C01810=1224.930,186.137,-55.083,-177.570,5.975,148.343
C01811=1224.935,185.867,-55.058,-177.573,5.973,148.343
C01812=1224.941,185.598,-55.033,-177.576,5.971,148.344
C01813=1224.945,185.328,-55.009,-177.578,5.969,148.344
C01814=1224.951,185.058,-54.984,-177.580,5.968,148.345
C01815=1224.955,184.810,-54.961,-177.584,5.967,148.345
C01816=1224.959,184.561,-54.938,-177.586,5.965,148.345
C01817=1224.964,184.311,-54.915,-177.589,5.963,148.346
C01818=1224.969,184.063,-54.893,-177.591,5.962,148.346
C01819=1224.974,183.814,-54.869,-177.594,5.960,148.347
C01820=1224.978,183.565,-54.846,-177.597,5.959,148.347
C01821=1224.982,183.316,-54.823,-177.599,5.958,148.348
C01822=1224.987,183.067,-54.800,-177.602,5.956,148.348
C01823=1224.992,182.819,-54.778,-177.604,5.954,148.348
C01824=1224.997,182.569,-54.755,-177.606,5.953,148.349
C01825=1225.002,182.320,-54.732,-177.609,5.952,148.349
C01826=1225.005,182.071,-54.709,-177.612,5.950,148.350
C01827=1225.011,181.823,-54.686,-177.614,5.949,148.350
C01828=1225.015,181.574,-54.664,-177.617,5.947,148.350
C01829=1225.020,181.324,-54.641,-177.620,5.945,148.351
C01830=1225.024,181.076,-54.618,-177.622,5.944,148.351
C01831=1225.029,180.827,-54.595,-177.625,5.943,148.352
C01832=1225.034,180.578,-54.572,-177.627,5.941,148.352
C01833=1225.038,180.329,-54.550,-177.629,5.940,148.352
C01834=1225.043,180.079,-54.527,-177.633,5.938,148.353
C01835=1225.048,179.831,-54.505,-177.635,5.936,148.353
C01836=1225.052,179.582,-54.481,-177.637,5.935,148.354
C01837=1225.057,179.333,-54.459,-177.640,5.934,148.354
C01838=1225.062,179.085,-54.436,-177.643,5.932,148.355
C01839=1225.066,178.835,-54.414,-177.645,5.931,148.355
C01840=1225.071,178.586,-54.391,-177.648,5.929,148.355
C01841=1225.075,178.338,-54.368,-177.650,5.928,148.356
C01842=1225.080,178.089,-54.346,-177.653,5.926,148.356
C01843=1225.084,177.840,-54.323,-177.656,5.925,148.357
C01844=1225.089,177.590,-54.300,-177.658,5.924,148.357
C01845=1225.094,177.342,-54.278,-177.660,5.922,148.357
C01846=1225.098,177.093,-54.256,-177.663,5.920,148.358
C01847=1225.103,176.844,-54.233,-177.666,5.920,148.358
C01848=1225.108,176.595,-54.211,-177.668,5.918,148.359
C01849=1225.112,176.346,-54.188,-177.671,5.916,148.359
C01850=1225.117,176.097,-54.166,-177.673,5.915,148.359
C01851=1225.122,175.848,-54.143,-177.676,5.913,148.360
C01852=1225.126,175.599,-54.120,-177.678,5.912,148.360
C01853=1225.131,175.350,-54.099,-177.681,5.911,148.361
C01854=1225.136,175.101,-54.075,-177.684,5.909,148.361
C01855=1225.140,174.852,-54.053,-177.686,5.908,148.362
C01856=1225.145,174.604,-54.030,-177.689,5.906,148.362
C01857=1225.150,174.354,-54.008,-177.691,5.904,148.362
C01858=1225.154,174.105,-53.986,-177.694,5.903,148.363
C01859=1225.159,173.857,-53.963,-177.697,5.902,148.363
C01860=1225.164,173.607,-53.941,-177.699,5.901,148.364
C01861=1225.168,173.359,-53.919,-177.701,5.899,148.364
C01862=1225.173,173.110,-53.896,-177.704,5.897,148.365
C01863=1225.177,172.860,-53.874,-177.707,5.897,148.365
C01864=1225.182,172.612,-53.852,-177.709,5.895,148.365
C01865=1225.187,172.363,-53.829,-177.712,5.893,148.366
C01866=1225.192,172.114,-53.807,-177.715,5.892,148.366
C01867=1225.196,171.865,-53.785,-177.717,5.890,148.367
C01868=1225.201,171.616,-53.762,-177.719,5.889,148.367
C01869=1225.206,171.367,-53.740,-177.722,5.888,148.368
C01870=1225.210,171.118,-53.718,-177.725,5.886,148.368
C01871=1225.214,170.870,-53.696,-177.727,5.885,148.369
C01872=1225.219,170.620,-53.673,-177.730,5.883,148.369
C01873=1225.224,170.371,-53.652,-177.732,5.882,148.369
C01874=1225.229,170.122,-53.630,-177.735,5.881,148.370
C01875=1225.233,169.873,-53.607,-177.737,5.880,148.370
C01876=1225.238,169.624,-53.584,-177.740,5.878,148.371
C01877=1225.242,169.375,-53.562,-177.743,5.876,148.371
C01878=1225.247,169.126,-53.541,-177.745,5.875,148.372
C01879=1225.252,168.877,-53.519,-177.748,5.874,148.372
C01880=1225.257,168.628,-53.496,-177.750,5.873,148.372
C01881=1225.261,168.379,-53.474,-177.753,5.871,148.373
C01882=1225.266,168.131,-53.452,-177.756,5.869,148.373
C01883=1225.270,167.881,-53.430,-177.758,5.868,148.374
C01884=1225.275,167.633,-53.408,-177.761,5.867,148.374
C01885=1225.280,167.383,-53.386,-177.763,5.866,148.375
C01886=1225.285,167.134,-53.364,-177.766,5.864,148.375
C01887=1225.289,166.885,-53.342,-177.768,5.863,148.376
C01888=1225.294,166.637,-53.320,-177.771,5.862,148.376
C01889=1225.298,166.387,-53.298,-177.774,5.860,148.376
C01890=1225.303,166.139,-53.276,-177.776,5.859,148.377
C01891=1225.308,165.889,-53.254,-177.779,5.857,148.377
C01892=1225.313,165.640,-53.232,-177.781,5.856,148.378
C01893=1225.317,165.392,-53.209,-177.784,5.854,148.378
C01894=1225.322,165.143,-53.188,-177.786,5.854,148.379
C01895=1225.326,164.894,-53.166,-177.789,5.852,148.379
C01896=1225.331,164.645,-53.144,-177.791,5.850,148.379
C01897=1225.335,164.396,-53.122,-177.794,5.849,148.380
C01898=1225.340,164.147,-53.100,-177.797,5.848,148.380
C01899=1225.345,163.898,-53.079,-177.799,5.847,148.381
C01900=1225.350,163.648,-53.057,-177.802,5.845,148.381
C01901=1225.355,163.399,-53.035,-177.804,5.844,148.382
C01902=1225.360,163.150,-53.013,-177.807,5.842,148.382
C01903=1225.364,162.901,-52.991,-177.809,5.842,148.383
C01904=1225.369,162.652,-52.969,-177.812,5.840,148.383
C01905=1225.374,162.403,-52.947,-177.815,5.838,148.384
C01906=1225.378,162.155,-52.926,-177.817,5.837,148.384
C01907=1225.383,161.905,-52.904,-177.820,5.836,148.384
C01908=1225.388,161.657,-52.882,-177.822,5.835,148.385
C01909=1225.392,161.407,-52.860,-177.825,5.833,148.385
C01910=1225.397,161.159,-52.838,-177.827,5.832,148.386
C01911=1225.402,160.910,-52.817,-177.830,5.830,148.386
C01912=1225.406,160.660,-52.795,-177.832,5.830,148.387
C01913=1225.411,160.412,-52.774,-177.835,5.828,148.387
C01914=1225.415,160.162,-52.752,-177.837,5.827,148.388
C01915=1225.421,159.893,-52.728,-177.840,5.825,148.388
C01916=1225.425,159.624,-52.705,-177.843,5.823,148.389
C01917=1225.431,159.355,-52.681,-177.846,5.822,148.389
C01918=1225.435,159.086,-52.659,-177.848,5.821,148.390
C01919=1225.440,158.837,-52.637,-177.851,5.819,148.390
C01920=1225.445,158.588,-52.615,-177.854,5.818,148.391
C01921=1225.449,158.339,-52.593,-177.856,5.817,148.391
C01922=1225.455,158.090,-52.572,-177.859,5.816,148.392
C01923=1225.459,157.841,-52.550,-177.861,5.814,148.392
C01924=1225.464,157.592,-52.529,-177.864,5.814,148.393
C01925=1225.469,157.343,-52.508,-177.867,5.812,148.393
C01926=1225.473,157.094,-52.486,-177.869,5.811,148.393
C01927=1225.478,156.845,-52.464,-177.872,5.809,148.394
C01928=1225.483,156.596,-52.442,-177.874,5.808,148.394
C01929=1225.487,156.347,-52.421,-177.877,5.806,148.395
C01930=1225.492,156.098,-52.400,-177.879,5.806,148.395
C01931=1225.497,155.849,-52.378,-177.882,5.804,148.396
C01932=1225.502,155.600,-52.357,-177.884,5.803,148.396
C01933=1225.506,155.351,-52.335,-177.887,5.801,148.397
C01934=1225.511,155.101,-52.314,-177.889,5.800,148.397
C01935=1225.516,154.853,-52.292,-177.893,5.799,148.398
C01936=1225.520,154.604,-52.271,-177.895,5.798,148.398
C01937=1225.525,154.355,-52.250,-177.897,5.796,148.398
C01938=1225.530,154.106,-52.228,-177.900,5.796,148.399
C01939=1225.534,153.856,-52.207,-177.903,5.794,148.399
C01940=1225.539,153.607,-52.185,-177.905,5.793,148.400
C01941=1225.544,153.359,-52.164,-177.908,5.791,148.400
C01942=1225.548,153.110,-52.143,-177.910,5.790,148.401
C01943=1225.553,152.860,-52.121,-177.913,5.789,148.401
C01944=1225.558,152.611,-52.100,-177.915,5.788,148.402
C01945=1225.563,152.362,-52.079,-177.918,5.786,148.402
C01946=1225.568,152.113,-52.058,-177.920,5.785,148.403
C01947=1225.571,151.864,-52.036,-177.923,5.783,148.403
C01948=1225.577,151.615,-52.015,-177.926,5.783,148.404
C01949=1225.581,151.366,-51.993,-177.928,5.781,148.404
C01950=1225.587,151.117,-51.972,-177.930,5.780,148.405
C01951=1225.591,150.869,-51.951,-177.934,5.779,148.405
C01952=1225.595,150.619,-51.930,-177.936,5.778,148.406
C01953=1225.600,150.369,-51.909,-177.939,5.776,148.406
C01954=1225.605,150.121,-51.888,-177.941,5.775,148.407
C01955=1225.610,149.872,-51.867,-177.944,5.773,148.407
C01956=1225.614,149.623,-51.845,-177.946,5.773,148.408
C01957=1225.619,149.373,-51.824,-177.949,5.771,148.408
C01958=1225.624,149.124,-51.804,-177.951,5.770,148.409
C01959=1225.629,148.876,-51.782,-177.954,5.769,148.409
C01960=1225.634,148.626,-51.761,-177.956,5.767,148.409
C01961=1225.637,148.377,-51.740,-177.959,5.767,148.410
C01962=1225.642,148.128,-51.719,-177.962,5.765,148.410
C01963=1225.648,147.879,-51.698,-177.964,5.764,148.411
C01964=1225.652,147.631,-51.677,-177.967,5.762,148.411
C01965=1225.657,147.381,-51.656,-177.969,5.761,148.412
C01966=1225.662,147.132,-51.635,-177.972,5.760,148.412
C01967=1225.666,146.883,-51.613,-177.974,5.759,148.413
C01968=1225.671,146.634,-51.592,-177.977,5.758,148.413
C01969=1225.675,146.385,-51.572,-177.979,5.757,148.414
C01970=1225.680,146.136,-51.551,-177.982,5.756,148.414
C01971=1225.685,145.887,-51.529,-177.985,5.754,148.415
C01972=1225.690,145.638,-51.509,-177.987,5.753,148.415
C01973=1225.695,145.389,-51.488,-177.990,5.752,148.416
C01974=1225.699,145.139,-51.467,-177.992,5.751,148.416
C01975=1225.704,144.890,-51.445,-177.995,5.749,148.417
C01976=1225.709,144.641,-51.424,-177.997,5.748,148.417
C01977=1225.713,144.392,-51.404,-178.000,5.748,148.418
C01978=1225.718,144.143,-51.383,-178.003,5.746,148.418
C01979=1225.723,143.894,-51.363,-178.005,5.745,148.418
C01980=1225.728,143.645,-51.341,-178.008,5.743,148.419
C01981=1225.732,143.396,-51.321,-178.010,5.742,148.419
C01982=1225.737,143.147,-51.300,-178.013,5.741,148.420
C01983=1225.741,142.897,-51.279,-178.015,5.740,148.420
C01984=1225.746,142.648,-51.258,-178.018,5.739,148.421
C01985=1225.751,142.399,-51.238,-178.020,5.737,148.421
C01986=1225.756,142.151,-51.216,-178.023,5.737,148.422
C01987=1225.760,141.902,-51.196,-178.026,5.735,148.422
C01988=1225.765,141.652,-51.175,-178.028,5.734,148.423
C01989=1225.770,141.403,-51.154,-178.031,5.732,148.424
C01990=1225.775,141.154,-51.133,-178.033,5.732,148.424
C01991=1225.779,140.905,-51.113,-178.036,5.731,148.425
C01992=1225.784,140.656,-51.092,-178.038,5.729,148.425
C01993=1225.789,140.407,-51.072,-178.041,5.728,148.426
C01994=1225.794,140.158,-51.051,-178.044,5.727,148.426
C01995=1225.798,139.909,-51.030,-178.046,5.726,148.427
C01996=1225.804,139.660,-51.009,-178.048,5.725,148.427
C01997=1225.808,139.411,-50.989,-178.052,5.724,148.428
C01998=1225.812,139.161,-50.968,-178.054,5.723,148.428
C01999=1225.817,138.912,-50.947,-178.056,5.721,148.428
C02000=1225.822,138.663,-50.927,-178.059,5.720,148.429
C02001=1225.827,138.414,-50.906,-178.061,5.719,148.429
C02002=1225.831,138.165,-50.885,-178.064,5.718,148.430
C02003=1225.836,137.915,-50.864,-178.066,5.717,148.430
C02004=1225.841,137.666,-50.844,-178.069,5.715,148.431
C02005=1225.845,137.417,-50.824,-178.072,5.714,148.431
C02006=1225.850,137.168,-50.803,-178.074,5.714,148.432
C02007=1225.855,136.919,-50.782,-178.077,5.712,148.432
C02008=1225.859,136.670,-50.762,-178.079,5.711,148.433
C02009=1225.864,136.421,-50.741,-178.082,5.709,148.433
C02010=1225.869,136.172,-50.721,-178.085,5.709,148.434
C02011=1225.874,135.922,-50.701,-178.087,5.708,148.434
C02012=1225.879,135.673,-50.680,-178.090,5.706,148.435
C02013=1225.883,135.424,-50.660,-178.092,5.705,148.435
C02014=1225.888,135.176,-50.640,-178.095,5.705,148.436
C02015=1225.893,134.927,-50.619,-178.097,5.703,148.436
C02016=1225.898,134.678,-50.598,-178.100,5.702,148.437
C02017=1225.903,134.428,-50.579,-178.103,5.700,148.437
C02018=1225.908,134.179,-50.558,-178.105,5.700,148.438
C02019=1225.912,133.910,-50.536,-178.108,5.698,148.439
C02020=1225.917,133.641,-50.514,-178.111,5.697,148.439
C02021=1225.923,133.373,-50.491,-178.114,5.696,148.440
C02022=1225.928,133.104,-50.470,-178.116,5.695,148.440
C02023=1225.933,132.855,-50.449,-178.119,5.693,148.441
C02024=1225.937,132.606,-50.429,-178.121,5.692,148.441
C02025=1225.942,132.357,-50.409,-178.124,5.692,148.442
C02026=1225.946,132.108,-50.389,-178.126,5.690,148.442
C02027=1225.952,131.858,-50.368,-178.129,5.689,148.443
C02028=1225.956,131.609,-50.348,-178.131,5.688,148.443
C02029=1225.961,131.360,-50.327,-178.134,5.687,148.444
C02030=1225.966,131.112,-50.308,-178.136,5.686,148.444
C02031=1225.971,130.862,-50.287,-178.139,5.685,148.445
C02032=1225.975,130.613,-50.267,-178.142,5.683,148.445
C02033=1225.980,130.364,-50.247,-178.144,5.683,148.446
C02034=1225.985,130.115,-50.227,-178.146,5.682,148.446
C02035=1225.989,129.866,-50.206,-178.150,5.680,148.447
C02036=1225.995,129.616,-50.186,-178.152,5.679,148.447
C02037=1225.999,129.367,-50.166,-178.155,5.678,148.448
C02038=1226.004,129.119,-50.146,-178.157,5.677,148.448
C02039=1226.009,128.869,-50.126,-178.160,5.676,148.449
C02040=1226.013,128.620,-50.106,-178.163,5.675,148.450
C02041=1226.018,128.371,-50.086,-178.165,5.674,148.450
C02042=1226.023,128.121,-50.065,-178.167,5.673,148.451
C02043=1226.028,127.873,-50.045,-178.170,5.672,148.451
C02044=1226.032,127.623,-50.025,-178.173,5.671,148.452
C02045=1226.037,127.375,-50.005,-178.175,5.670,148.452
C02046=1226.042,127.125,-49.985,-178.178,5.668,148.453
C02047=1226.047,126.876,-49.965,-178.180,5.667,148.453
C02048=1226.051,126.627,-49.945,-178.183,5.667,148.454
C02049=1226.056,126.378,-49.925,-178.185,5.665,148.454
C02050=1226.060,126.128,-49.905,-178.188,5.664,148.455
C02051=1226.066,125.880,-49.885,-178.190,5.663,148.455
C02052=1226.071,125.630,-49.865,-178.193,5.662,148.456
C02053=1226.075,125.381,-49.845,-178.195,5.661,148.456
C02054=1226.080,125.131,-49.825,-178.198,5.660,148.457
C02055=1226.085,124.883,-49.805,-178.201,5.660,148.457
C02056=1226.090,124.634,-49.785,-178.203,5.658,148.458
C02057=1226.094,124.385,-49.765,-178.206,5.657,148.458
C02058=1226.099,124.135,-49.745,-178.208,5.656,148.459
C02059=1226.104,123.886,-49.725,-178.211,5.655,148.459
C02060=1226.108,123.637,-49.705,-178.213,5.654,148.460
C02061=1226.114,123.388,-49.686,-178.216,5.653,148.461
C02062=1226.118,123.139,-49.666,-178.219,5.651,148.461
C02063=1226.123,122.889,-49.646,-178.221,5.651,148.462
C02064=1226.127,122.640,-49.626,-178.223,5.650,148.462
C02065=1226.133,122.391,-49.606,-178.226,5.648,148.463
C02066=1226.137,122.142,-49.587,-178.229,5.648,148.463
C02067=1226.142,121.893,-49.566,-178.231,5.647,148.464
C02068=1226.147,121.643,-49.547,-178.234,5.646,148.464
C02069=1226.152,121.394,-49.527,-178.236,5.644,148.465
C02070=1226.156,121.146,-49.507,-178.239,5.644,148.465
C02071=1226.161,120.896,-49.487,-178.241,5.643,148.466
C02072=1226.166,120.646,-49.468,-178.244,5.641,148.466
C02073=1226.171,120.398,-49.448,-178.247,5.641,148.467
C02074=1226.176,120.149,-49.428,-178.249,5.640,148.467
C02075=1226.180,119.899,-49.408,-178.252,5.638,148.468
C02076=1226.186,119.650,-49.389,-178.254,5.637,148.468
C02077=1226.189,119.401,-49.369,-178.257,5.637,148.469
C02078=1226.194,119.152,-49.350,-178.259,5.636,148.469
C02079=1226.199,118.902,-49.330,-178.262,5.634,148.470
C02080=1226.204,118.653,-49.311,-178.265,5.634,148.471
C02081=1226.209,118.405,-49.290,-178.267,5.633,148.471
C02082=1226.213,118.155,-49.271,-178.270,5.631,148.472
C02083=1226.219,117.906,-49.251,-178.272,5.630,148.472
C02084=1226.223,117.657,-49.232,-178.275,5.630,148.473
C02085=1226.228,117.407,-49.212,-178.277,5.629,148.473
C02086=1226.233,117.159,-49.193,-178.280,5.627,148.474
C02087=1226.237,116.909,-49.173,-178.283,5.627,148.474
C02088=1226.242,116.660,-49.153,-178.285,5.626,148.475
C02089=1226.247,116.411,-49.134,-178.288,5.625,148.476
C02090=1226.252,116.161,-49.114,-178.290,5.623,148.476
C02091=1226.257,115.912,-49.095,-178.293,5.623,148.477
C02092=1226.262,115.663,-49.075,-178.295,5.622,148.477
C02093=1226.266,115.414,-49.056,-178.298,5.620,148.478
C02094=1226.271,115.165,-49.036,-178.301,5.620,148.478
C02095=1226.276,114.916,-49.017,-178.303,5.619,148.479
C02096=1226.281,114.666,-48.997,-178.305,5.618,148.479
C02097=1226.286,114.418,-48.978,-178.309,5.617,148.480
C02098=1226.290,114.168,-48.959,-178.311,5.616,148.480
C02099=1226.295,113.919,-48.939,-178.313,5.615,148.481
C02100=1226.300,113.670,-48.920,-178.315,5.614,148.481
C02101=1226.305,113.420,-48.900,-178.319,5.613,148.482
C02102=1226.309,113.171,-48.881,-178.321,5.612,148.483
C02103=1226.314,112.922,-48.862,-178.323,5.611,148.483
C02104=1226.319,112.673,-48.842,-178.326,5.610,148.484
C02105=1226.324,112.424,-48.823,-178.329,5.609,148.484
C02106=1226.328,112.174,-48.804,-178.331,5.608,148.485
C02107=1226.333,111.925,-48.784,-178.334,5.607,148.485
C02108=1226.338,111.676,-48.765,-178.336,5.606,148.486
C02109=1226.343,111.426,-48.745,-178.339,5.605,148.486
C02110=1226.348,111.178,-48.726,-178.341,5.604,148.487
C02111=1226.353,110.928,-48.707,-178.344,5.603,148.487
C02112=1226.358,110.679,-48.687,-178.347,5.603,148.488
C02113=1226.362,110.430,-48.668,-178.349,5.601,148.489
C02114=1226.367,110.181,-48.649,-178.352,5.600,148.489
C02115=1226.372,109.932,-48.629,-178.354,5.600,148.490
C02116=1226.376,109.682,-48.610,-178.357,5.599,148.490
C02117=1226.382,109.433,-48.592,-178.359,5.598,148.491
C02118=1226.386,109.183,-48.572,-178.362,5.596,148.491
C02119=1226.391,108.935,-48.553,-178.364,5.596,148.492
C02120=1226.396,108.685,-48.534,-178.367,5.595,148.493
C02121=1226.401,108.436,-48.514,-178.369,5.594,148.493
C02122=1226.405,108.187,-48.495,-178.372,5.593,148.494
C02123=1226.411,107.919,-48.475,-178.375,5.592,148.494
C02124=1226.416,107.650,-48.454,-178.378,5.591,148.495
C02125=1226.421,107.382,-48.434,-178.380,5.590,148.495
C02126=1226.426,107.113,-48.413,-178.383,5.589,148.496
C02127=1226.431,106.864,-48.395,-178.386,5.588,148.497
C02128=1226.436,106.615,-48.375,-178.389,5.587,148.497
C02129=1226.440,106.366,-48.356,-178.391,5.586,148.498
C02130=1226.445,106.116,-48.337,-178.393,5.585,148.498
C02131=1226.451,105.867,-48.318,-178.396,5.584,148.499
C02132=1226.455,105.618,-48.299,-178.398,5.584,148.499
C02133=1226.460,105.369,-48.280,-178.401,5.582,148.500
C02134=1226.464,105.120,-48.261,-178.404,5.581,148.500
C02135=1226.470,104.870,-48.242,-178.406,5.581,148.501
C02136=1226.474,104.621,-48.223,-178.409,5.580,148.502
C02137=1226.479,104.372,-48.204,-178.411,5.579,148.502
C02138=1226.484,104.122,-48.184,-178.414,5.578,148.503
C02139=1226.489,103.873,-48.166,-178.417,5.577,148.503
C02140=1226.494,103.624,-48.146,-178.419,5.576,148.504
C02141=1226.498,103.375,-48.128,-178.421,5.576,148.504
C02142=1226.503,103.125,-48.109,-178.424,5.575,148.505
C02143=1226.508,102.876,-48.090,-178.427,5.573,148.505
C02144=1226.513,102.628,-48.071,-178.429,5.573,148.506
C02145=1226.518,102.378,-48.052,-178.432,5.572,148.507
C02146=1226.523,102.129,-48.033,-178.434,5.571,148.507
C02147=1226.527,101.879,-48.015,-178.437,5.570,148.508
C02148=1226.533,101.630,-47.995,-178.440,5.569,148.508
C02149=1226.537,101.381,-47.976,-178.442,5.568,148.509
C02150=1226.541,101.132,-47.958,-178.445,5.567,148.510
C02151=1226.547,100.883,-47.939,-178.447,5.567,148.510
C02152=1226.551,100.633,-47.921,-178.449,5.566,148.511
C02153=1226.556,100.384,-47.901,-178.453,5.564,148.511
C02154=1226.561,100.134,-47.883,-178.455,5.564,148.512
C02155=1226.566,99.885,-47.864,-178.457,5.563,148.512
C02156=1226.571,99.637,-47.845,-178.460,5.562,148.513
C02157=1226.575,99.387,-47.827,-178.463,5.562,148.514
C02158=1226.580,99.138,-47.808,-178.465,5.561,148.514
C02159=1226.585,98.888,-47.789,-178.468,5.559,148.515
C02160=1226.590,98.639,-47.770,-178.470,5.559,148.515
C02161=1226.595,98.390,-47.752,-178.473,5.558,148.516
C02162=1226.599,98.141,-47.733,-178.475,5.557,148.516
C02163=1226.605,97.891,-47.714,-178.478,5.557,148.517
C02164=1226.609,97.643,-47.696,-178.480,5.556,148.517
C02165=1226.614,97.393,-47.677,-178.483,5.554,148.518
C02166=1226.619,97.143,-47.659,-178.486,5.554,148.519
C02167=1226.624,96.895,-47.640,-178.488,5.553,148.519
C02168=1226.629,96.645,-47.621,-178.490,5.552,148.520
C02169=1226.633,96.396,-47.602,-178.493,5.551,148.520
C02170=1226.638,96.146,-47.584,-178.495,5.550,148.521
C02171=1226.643,95.897,-47.565,-178.498,5.549,148.521
C02172=1226.648,95.648,-47.547,-178.501,5.548,148.522
C02173=1226.653,95.399,-47.529,-178.504,5.548,148.523
C02174=1226.658,95.149,-47.509,-178.506,5.547,148.523
C02175=1226.663,94.900,-47.491,-178.508,5.546,148.524
C02176=1226.667,94.651,-47.473,-178.511,5.546,148.525
C02177=1226.671,94.402,-47.454,-178.514,5.544,148.525
C02178=1226.677,94.152,-47.435,-178.516,5.543,148.526
C02179=1226.682,93.903,-47.417,-178.519,5.543,148.526
C02180=1226.686,93.654,-47.398,-178.521,5.542,148.527
C02181=1226.692,93.404,-47.380,-178.524,5.541,148.527
C02182=1226.697,93.155,-47.362,-178.526,5.540,148.528
C02183=1226.701,92.906,-47.343,-178.529,5.540,148.529
C02184=1226.706,92.657,-47.325,-178.532,5.538,148.529
C02185=1226.711,92.407,-47.306,-178.534,5.537,148.530
C02186=1226.716,92.159,-47.288,-178.537,5.537,148.530
C02187=1226.720,91.909,-47.269,-178.539,5.536,148.531
C02188=1226.725,91.660,-47.251,-178.542,5.535,148.531
C02189=1226.730,91.411,-47.233,-178.544,5.535,148.532
C02190=1226.735,91.162,-47.214,-178.546,5.534,148.532
C02191=1226.740,90.912,-47.196,-178.549,5.533,148.533
C02192=1226.744,90.663,-47.178,-178.552,5.532,148.534
C02193=1226.749,90.413,-47.160,-178.555,5.531,148.534
C02194=1226.754,90.164,-47.142,-178.557,5.530,148.535
C02195=1226.759,89.915,-47.122,-178.560,5.530,148.535
C02196=1226.764,89.665,-47.104,-178.562,5.529,148.536
C02197=1226.769,89.416,-47.086,-178.564,5.528,148.537
C02198=1226.774,89.167,-47.068,-178.567,5.527,148.537
C02199=1226.778,88.917,-47.050,-178.570,5.527,148.538
C02200=1226.783,88.668,-47.032,-178.573,5.525,148.538
C02201=1226.789,88.419,-47.013,-178.575,5.524,148.539
C02202=1226.793,88.170,-46.994,-178.577,5.524,148.540
C02203=1226.798,87.921,-46.977,-178.580,5.523,148.540
C02204=1226.802,87.671,-46.958,-178.583,5.523,148.541
C02205=1226.807,87.422,-46.940,-178.585,5.522,148.541
C02206=1226.812,87.173,-46.922,-178.587,5.521,148.542
C02207=1226.817,86.923,-46.904,-178.590,5.521,148.543
C02208=1226.822,86.674,-46.886,-178.592,5.520,148.543
C02209=1226.827,86.424,-46.867,-178.595,5.518,148.544
C02210=1226.832,86.175,-46.849,-178.598,5.518,148.544
C02211=1226.837,85.926,-46.831,-178.601,5.517,148.545
C02212=1226.842,85.677,-46.813,-178.603,5.516,148.545
C02213=1226.847,85.427,-46.795,-178.605,5.515,148.546
C02214=1226.852,85.178,-46.777,-178.608,5.515,148.547
C02215=1226.856,84.928,-46.759,-178.611,5.514,148.547
C02216=1226.861,84.679,-46.741,-178.613,5.513,148.548
C02217=1226.866,84.430,-46.723,-178.615,5.513,148.548
C02218=1226.871,84.181,-46.705,-178.619,5.511,148.549
C02219=1226.876,83.932,-46.687,-178.621,5.511,148.550
C02220=1226.881,83.682,-46.669,-178.623,5.510,148.550
C02221=1226.886,83.433,-46.651,-178.626,5.509,148.551
C02222=1226.890,83.183,-46.633,-178.629,5.509,148.551
C02223=1226.895,82.934,-46.615,-178.631,5.508,148.552
C02224=1226.900,82.685,-46.597,-178.633,5.507,148.553
C02225=1226.905,82.436,-46.579,-178.636,5.506,148.553
C02226=1226.909,82.187,-46.561,-178.639,5.506,148.554
C02227=1226.915,81.918,-46.542,-178.641,5.505,148.555
C02228=1226.920,81.650,-46.522,-178.644,5.504,148.555
C02229=1226.926,81.381,-46.503,-178.647,5.503,148.556
C02230=1226.931,81.113,-46.483,-178.650,5.503,148.556
C02231=1226.936,80.864,-46.465,-178.652,5.502,148.557
C02232=1226.941,80.614,-46.447,-178.654,5.501,148.558
C02233=1226.945,80.366,-46.430,-178.657,5.500,148.558
C02234=1226.950,80.116,-46.412,-178.660,5.499,148.559
C02235=1226.955,79.867,-46.395,-178.663,5.498,148.560
C02236=1226.960,79.617,-46.377,-178.665,5.498,148.560
C02237=1226.964,79.368,-46.358,-178.668,5.497,148.561
C02238=1226.969,79.118,-46.340,-178.670,5.496,148.561
C02239=1226.974,78.869,-46.323,-178.673,5.496,148.562
C02240=1226.979,78.620,-46.305,-178.675,5.495,148.562
C02241=1226.984,78.370,-46.287,-178.678,5.494,148.563
C02242=1226.989,78.121,-46.269,-178.680,5.494,148.564
C02243=1226.994,77.872,-46.251,-178.683,5.493,148.564
C02244=1226.999,77.623,-46.233,-178.685,5.492,148.565
C02245=1227.003,77.373,-46.217,-178.688,5.491,148.565
C02246=1227.008,77.124,-46.199,-178.690,5.491,148.566
C02247=1227.013,76.875,-46.181,-178.693,5.490,148.567
C02248=1227.018,76.626,-46.163,-178.696,5.490,148.567
C02249=1227.023,76.376,-46.145,-178.698,5.489,148.568
C02250=1227.028,76.127,-46.127,-178.701,5.487,148.568
C02251=1227.033,75.878,-46.110,-178.703,5.487,148.569
C02252=1227.038,75.628,-46.093,-178.706,5.486,148.570
C02253=1227.043,75.379,-46.075,-178.708,5.485,148.570
C02254=1227.047,75.130,-46.057,-178.711,5.485,148.571
C02255=1227.053,74.880,-46.040,-178.714,5.484,148.572
C02256=1227.058,74.631,-46.022,-178.716,5.483,148.572
C02257=1227.062,74.382,-46.004,-178.719,5.483,148.573
C02258=1227.067,74.132,-45.987,-178.721,5.482,148.573
C02259=1227.072,73.883,-45.969,-178.724,5.481,148.574
C02260=1227.077,73.634,-45.951,-178.726,5.481,148.575
C02261=1227.082,73.384,-45.934,-178.729,5.480,148.575
C02262=1227.086,73.135,-45.916,-178.731,5.480,148.576
C02263=1227.091,72.885,-45.899,-178.734,5.479,148.576
C02264=1227.096,72.636,-45.881,-178.736,5.478,148.577
C02265=1227.101,72.387,-45.863,-178.739,5.477,148.578
C02266=1227.106,72.137,-45.846,-178.741,5.477,148.578
C02267=1227.111,71.888,-45.828,-178.744,5.476,148.579
C02268=1227.116,71.638,-45.811,-178.746,5.475,148.579
C02269=1227.121,71.389,-45.793,-178.749,5.475,148.580
C02270=1227.125,71.140,-45.777,-178.751,5.474,148.581
C02271=1227.130,70.891,-45.759,-178.754,5.474,148.581
C02272=1227.135,70.641,-45.741,-178.756,5.473,148.582
C02273=1227.140,70.392,-45.724,-178.759,5.472,148.582
C02274=1227.145,70.142,-45.707,-178.762,5.471,148.583
C02275=1227.150,69.894,-45.689,-178.765,5.470,148.584
C02276=1227.155,69.644,-45.672,-178.767,5.470,148.584
C02277=1227.160,69.395,-45.654,-178.770,5.469,148.585
C02278=1227.165,69.145,-45.637,-178.772,5.468,148.586
C02279=1227.170,68.896,-45.619,-178.775,5.467,148.586
C02280=1227.174,68.647,-45.603,-178.777,5.467,148.587
C02281=1227.179,68.397,-45.585,-178.780,5.466,148.588
C02282=1227.184,68.148,-45.567,-178.783,5.466,148.588
C02283=1227.189,67.898,-45.551,-178.785,5.465,148.589
C02284=1227.194,67.649,-45.533,-178.787,5.464,148.589
C02285=1227.198,67.399,-45.516,-178.790,5.464,148.590
C02286=1227.204,67.151,-45.498,-178.793,5.463,148.591
C02287=1227.209,66.901,-45.481,-178.795,5.462,148.591
C02288=1227.213,66.652,-45.464,-178.797,5.461,148.592
C02289=1227.218,66.403,-45.446,-178.800,5.461,148.592
C02290=1227.224,66.153,-45.429,-178.803,5.460,148.593
C02291=1227.228,65.904,-45.412,-178.805,5.460,148.594
C02292=1227.233,65.654,-45.395,-178.808,5.459,148.594
C02293=1227.237,65.405,-45.378,-178.811,5.459,148.595
C02294=1227.243,65.156,-45.360,-178.813,5.458,148.595
C02295=1227.247,64.907,-45.344,-178.815,5.457,148.596
C02296=1227.253,64.657,-45.326,-178.818,5.456,148.597
C02297=1227.258,64.407,-45.309,-178.821,5.456,148.597
C02298=1227.262,64.158,-45.292,-178.823,5.455,148.598
C02299=1227.267,63.908,-45.274,-178.826,5.455,148.599
C02300=1227.272,63.660,-45.258,-178.828,5.454,148.599
C02301=1227.277,63.410,-45.240,-178.831,5.453,148.600
C02302=1227.282,63.161,-45.223,-178.833,5.453,148.601
C02303=1227.287,62.911,-45.206,-178.836,5.452,148.601
C02304=1227.291,62.662,-45.189,-178.839,5.451,148.602
C02305=1227.296,62.412,-45.172,-178.841,5.451,148.602
C02306=1227.301,62.164,-45.155,-178.843,5.450,148.603
C02307=1227.307,61.914,-45.138,-178.846,5.449,148.604
C02308=1227.311,61.664,-45.121,-178.849,5.449,148.604
C02309=1227.316,61.415,-45.104,-178.851,5.448,148.605
C02310=1227.321,61.166,-45.087,-178.854,5.448,148.606
C02311=1227.326,60.917,-45.070,-178.856,5.447,148.606
C02312=1227.331,60.667,-45.053,-178.859,5.446,148.607
C02313=1227.336,60.417,-45.036,-178.861,5.446,148.607
C02314=1227.341,60.168,-45.019,-178.864,5.445,148.608
C02315=1227.346,59.919,-45.002,-178.866,5.444,148.609
C02316=1227.351,59.670,-44.985,-178.869,5.445,148.609
C02317=1227.356,59.420,-44.968,-178.871,5.444,148.610
C02318=1227.360,59.171,-44.951,-178.873,5.443,148.611
C02319=1227.366,58.922,-44.934,-178.876,5.443,148.611
C02320=1227.371,58.672,-44.917,-178.879,5.442,148.612
C02321=1227.375,58.423,-44.901,-178.881,5.441,148.613
C02322=1227.380,58.173,-44.883,-178.884,5.441,148.613
C02323=1227.385,57.924,-44.867,-178.886,5.440,148.614
C02324=1227.391,57.674,-44.850,-178.889,5.439,148.614
C02325=1227.395,57.425,-44.832,-178.891,5.439,148.615
C02326=1227.399,57.176,-44.816,-178.894,5.438,148.616
C02327=1227.405,56.927,-44.799,-178.897,5.438,148.616
C02328=1227.409,56.677,-44.782,-178.899,5.437,148.617
C02329=1227.415,56.428,-44.765,-178.902,5.436,148.618
C02330=1227.419,56.178,-44.748,-178.904,5.436,148.618
C02331=1227.424,55.910,-44.731,-178.907,5.435,148.619
C02332=1227.430,55.641,-44.713,-178.910,5.435,148.620
C02333=1227.435,55.373,-44.695,-178.912,5.434,148.620
C02334=1227.441,55.104,-44.676,-178.915,5.434,148.621
C02335=1227.446,54.855,-44.660,-178.918,5.433,148.622
C02336=1227.450,54.606,-44.643,-178.920,5.432,148.622
C02337=1227.456,54.356,-44.626,-178.923,5.432,148.623
C02338=1227.461,54.107,-44.610,-178.925,5.431,148.623
C02339=1227.465,53.858,-44.593,-178.928,5.430,148.624
C02340=1227.470,53.608,-44.576,-178.930,5.430,148.625
C02341=1227.475,53.359,-44.559,-178.933,5.429,148.625
C02342=1227.480,53.110,-44.543,-178.936,5.429,148.626
C02343=1227.485,52.860,-44.525,-178.938,5.428,148.627
C02344=1227.490,52.611,-44.509,-178.941,5.428,148.627
C02345=1227.495,52.361,-44.493,-178.943,5.427,148.628
C02346=1227.499,52.111,-44.477,-178.946,5.426,148.629
C02347=1227.505,51.862,-44.460,-178.948,5.425,148.629
C02348=1227.510,51.613,-44.443,-178.951,5.425,148.630
C02349=1227.514,51.363,-44.426,-178.954,5.424,148.631
C02350=1227.519,51.115,-44.410,-178.956,5.424,148.631
C02351=1227.525,50.865,-44.393,-178.958,5.424,148.632
C02352=1227.529,50.615,-44.377,-178.961,5.423,148.633
C02353=1227.534,50.366,-44.360,-178.963,5.423,148.633
C02354=1227.539,50.116,-44.344,-178.966,5.422,148.634
C02355=1227.545,49.867,-44.327,-178.968,5.421,148.634
C02356=1227.549,49.618,-44.310,-178.971,5.421,148.635
C02357=1227.554,49.368,-44.294,-178.974,5.420,148.636
C02358=1227.559,49.119,-44.278,-178.976,5.420,148.636
C02359=1227.564,48.869,-44.261,-178.979,5.419,148.637
C02360=1227.569,48.620,-44.244,-178.981,5.419,148.638
C02361=1227.574,48.371,-44.228,-178.984,5.418,148.638
C02362=1227.579,48.121,-44.212,-178.986,5.417,148.639
C02363=1227.584,47.872,-44.195,-178.989,5.417,148.639
C02364=1227.588,47.622,-44.179,-178.992,5.416,148.640
C02365=1227.593,47.374,-44.162,-178.994,5.416,148.641
C02366=1227.599,47.123,-44.146,-178.996,5.416,148.641
C02367=1227.603,46.874,-44.129,-178.999,5.415,148.642
C02368=1227.608,46.625,-44.113,-179.002,5.414,148.643
C02369=1227.613,46.375,-44.097,-179.004,5.414,148.643
C02370=1227.618,46.126,-44.081,-179.006,5.413,148.644
C02371=1227.623,45.877,-44.064,-179.009,5.412,148.645
C02372=1227.628,45.628,-44.048,-179.012,5.412,148.645
C02373=1227.633,45.377,-44.031,-179.014,5.411,148.646
C02374=1227.638,45.128,-44.015,-179.017,5.411,148.647
C02375=1227.643,44.879,-43.999,-179.019,5.410,148.647
C02376=1227.648,44.629,-43.982,-179.022,5.410,148.648
C02377=1227.653,44.380,-43.966,-179.024,5.410,148.649
C02378=1227.658,44.130,-43.950,-179.027,5.409,148.649
C02379=1227.663,43.881,-43.934,-179.029,5.408,148.650
C02380=1227.667,43.632,-43.917,-179.032,5.408,148.650
C02381=1227.672,43.383,-43.901,-179.034,5.407,148.651
C02382=1227.677,43.133,-43.885,-179.037,5.407,148.652
C02383=1227.682,42.884,-43.869,-179.040,5.406,148.652
C02384=1227.687,42.634,-43.853,-179.042,5.406,148.653
C02385=1227.693,42.384,-43.836,-179.045,5.405,148.654
C02386=1227.697,42.135,-43.820,-179.047,5.405,148.654
C02387=1227.702,41.886,-43.803,-179.050,5.405,148.655
C02388=1227.707,41.636,-43.787,-179.052,5.404,148.656
C02389=1227.712,41.387,-43.771,-179.055,5.404,148.656
C02390=1227.717,41.137,-43.755,-179.057,5.403,148.657
C02391=1227.722,40.888,-43.739,-179.060,5.402,148.658
C02392=1227.727,40.638,-43.723,-179.062,5.402,148.658
C02393=1227.732,40.390,-43.707,-179.065,5.401,148.659
C02394=1227.737,40.139,-43.691,-179.068,5.400,148.660
C02395=1227.742,39.891,-43.674,-179.070,5.400,148.660
C02396=1227.747,39.641,-43.658,-179.072,5.400,148.661
C02397=1227.752,39.392,-43.642,-179.075,5.400,148.662
C02398=1227.757,39.142,-43.626,-179.077,5.399,148.662
C02399=1227.762,38.893,-43.610,-179.080,5.398,148.663
C02400=1227.766,38.643,-43.594,-179.083,5.398,148.664
C02401=1227.772,38.393,-43.578,-179.085,5.397,148.664
C02402=1227.777,38.145,-43.562,-179.088,5.396,148.665
C02403=1227.782,37.894,-43.546,-179.090,5.396,148.665
C02404=1227.786,37.646,-43.530,-179.092,5.396,148.666
C02405=1227.791,37.396,-43.514,-179.095,5.396,148.667
C02406=1227.796,37.146,-43.499,-179.098,5.395,148.667
C02407=1227.801,36.897,-43.482,-179.100,5.394,148.668
C02408=1227.806,36.648,-43.467,-179.103,5.394,148.669
C02409=1227.811,36.399,-43.450,-179.105,5.393,148.670
C02410=1227.816,36.149,-43.434,-179.108,5.393,148.670
C02411=1227.821,35.899,-43.419,-179.111,5.392,148.671
C02412=1227.826,35.650,-43.402,-179.113,5.393,148.672
C02413=1227.831,35.400,-43.386,-179.115,5.392,148.672
C02414=1227.837,35.151,-43.371,-179.118,5.391,148.673
C02415=1227.840,34.902,-43.355,-179.120,5.390,148.673
C02416=1227.846,34.652,-43.339,-179.123,5.390,148.674
C02417=1227.851,34.402,-43.323,-179.126,5.389,148.675
C02418=1227.856,34.153,-43.308,-179.128,5.389,148.675
C02419=1227.861,33.904,-43.291,-179.130,5.389,148.676
C02420=1227.866,33.654,-43.275,-179.133,5.389,148.677
C02421=1227.871,33.405,-43.260,-179.136,5.388,148.677
C02422=1227.875,33.155,-43.244,-179.138,5.387,148.678
C02423=1227.880,32.906,-43.228,-179.141,5.387,148.679
C02424=1227.886,32.657,-43.213,-179.143,5.386,148.679
C02425=1227.890,32.407,-43.197,-179.146,5.386,148.680
C02426=1227.896,32.158,-43.180,-179.148,5.386,148.681
C02427=1227.901,31.908,-43.165,-179.150,5.385,148.681
C02428=1227.905,31.659,-43.149,-179.153,5.385,148.682
C02429=1227.910,31.409,-43.134,-179.156,5.384,148.683
C02430=1227.916,31.160,-43.118,-179.158,5.383,148.683
C02431=1227.920,30.910,-43.101,-179.161,5.383,148.684
C02432=1227.926,30.661,-43.086,-179.164,5.382,148.685
C02433=1227.930,30.412,-43.071,-179.166,5.383,148.685
C02434=1227.935,30.162,-43.055,-179.168,5.382,148.686
C02435=1227.941,29.893,-43.038,-179.171,5.382,148.687
C02436=1227.946,29.625,-43.021,-179.174,5.381,148.687
C02437=1227.951,29.357,-43.004,-179.177,5.381,148.688
C02438=1227.957,29.088,-42.987,-179.179,5.380,148.689
C02439=1227.961,28.838,-42.972,-179.182,5.380,148.690
C02440=1227.967,28.589,-42.956,-179.185,5.379,148.690
C02441=1227.971,28.339,-42.941,-179.187,5.378,148.691
C02442=1227.976,28.089,-42.925,-179.189,5.378,148.691
C02443=1227.982,27.840,-42.909,-179.191,5.378,148.692
C02444=1227.987,27.591,-42.894,-179.194,5.377,148.693
C02445=1227.992,27.341,-42.879,-179.197,5.377,148.693
C02446=1227.996,27.091,-42.863,-179.199,5.376,148.694
C02447=1228.002,26.842,-42.847,-179.202,5.376,148.695
C02448=1228.006,26.593,-42.832,-179.204,5.376,148.695
C02449=1228.011,26.343,-42.816,-179.207,5.375,148.696
C02450=1228.016,26.094,-42.800,-179.209,5.375,148.697
C02451=1228.021,25.845,-42.785,-179.212,5.374,148.698
C02452=1228.026,25.596,-42.769,-179.215,5.374,148.698
C02453=1228.031,25.345,-42.753,-179.217,5.373,148.699
C02454=1228.036,25.096,-42.738,-179.219,5.374,148.700
C02455=1228.041,24.847,-42.723,-179.222,5.373,148.700
C02456=1228.047,24.598,-42.707,-179.225,5.372,148.701
C02457=1228.051,24.348,-42.692,-179.227,5.372,148.702
C02458=1228.056,24.098,-42.677,-179.230,5.371,148.702
C02459=1228.062,23.848,-42.662,-179.233,5.371,148.703
C02460=1228.066,23.599,-42.647,-179.235,5.371,148.704
C02461=1228.072,23.350,-42.631,-179.237,5.370,148.704
C02462=1228.076,23.100,-42.616,-179.240,5.370,148.705
C02463=1228.081,22.851,-42.600,-179.242,5.369,148.705
C02464=1228.087,22.601,-42.584,-179.245,5.369,148.706
C02465=1228.091,22.352,-42.569,-179.247,5.369,148.707
C02466=1228.096,22.102,-42.553,-179.250,5.368,148.708
C02467=1228.101,21.853,-42.538,-179.252,5.368,148.708
C02468=1228.106,21.604,-42.523,-179.255,5.367,148.709
C02469=1228.111,21.354,-42.507,-179.257,5.367,148.710
C02470=1228.116,21.105,-42.492,-179.260,5.367,148.710
C02471=1228.121,20.854,-42.477,-179.262,5.366,148.711
C02472=1228.126,20.605,-42.462,-179.265,5.366,148.712
C02473=1228.131,20.356,-42.446,-179.268,5.365,148.712
C02474=1228.136,20.107,-42.431,-179.270,5.365,148.713
C02475=1228.141,19.857,-42.416,-179.272,5.365,148.714
C02476=1228.146,19.608,-42.401,-179.275,5.364,148.714
C02477=1228.151,19.357,-42.386,-179.278,5.364,148.715
C02478=1228.156,19.108,-42.371,-179.280,5.363,148.716
C02479=1228.161,18.859,-42.355,-179.283,5.363,148.716
C02480=1228.166,18.610,-42.339,-179.285,5.363,148.717
C02481=1228.171,18.361,-42.324,-179.288,5.363,148.718
C02482=1228.177,18.110,-42.310,-179.290,5.362,148.718
C02483=1228.181,17.861,-42.294,-179.293,5.361,148.719
C02484=1228.185,17.612,-42.279,-179.295,5.361,148.720
C02485=1228.191,17.362,-42.264,-179.298,5.361,148.720
C02486=1228.196,17.112,-42.249,-179.300,5.361,148.721
C02487=1228.201,16.863,-42.234,-179.303,5.360,148.722
C02488=1228.206,16.614,-42.219,-179.305,5.359,148.722
C02489=1228.211,16.365,-42.203,-179.308,5.359,148.723
C02490=1228.216,16.115,-42.189,-179.310,5.359,148.724
C02491=1228.221,15.865,-42.173,-179.312,5.358,148.724
C02492=1228.226,15.616,-42.158,-179.315,5.358,148.725
C02493=1228.231,15.366,-42.143,-179.318,5.357,148.726
C02494=1228.236,15.117,-42.128,-179.320,5.357,148.726
C02495=1228.241,14.867,-42.113,-179.322,5.357,148.727
C02496=1228.246,14.617,-42.098,-179.325,5.357,148.728
C02497=1228.251,14.368,-42.083,-179.328,5.356,148.728
C02498=1228.256,14.119,-42.068,-179.330,5.355,148.729
C02499=1228.261,13.869,-42.053,-179.332,5.356,148.730
C02500=1228.267,13.620,-42.038,-179.335,5.355,148.731
C02501=1228.271,13.370,-42.022,-179.338,5.355,148.731
C02502=1228.276,13.120,-42.008,-179.340,5.354,148.732
C02503=1228.281,12.871,-41.993,-179.343,5.354,148.733
C02504=1228.286,12.622,-41.978,-179.345,5.354,148.733
C02505=1228.291,12.372,-41.963,-179.348,5.353,148.734
C02506=1228.296,12.123,-41.948,-179.350,5.353,148.735
C02507=1228.301,11.873,-41.933,-179.353,5.352,148.735
C02508=1228.306,11.624,-41.918,-179.355,5.353,148.736
C02509=1228.311,11.374,-41.904,-179.358,5.352,148.737
C02510=1228.316,11.125,-41.889,-179.360,5.352,148.737
C02511=1228.321,10.875,-41.873,-179.363,5.351,148.738
C02512=1228.326,10.626,-41.859,-179.366,5.350,148.739
C02513=1228.331,10.377,-41.844,-179.368,5.351,148.739
C02514=1228.337,10.127,-41.829,-179.370,5.350,148.740
C02515=1228.341,9.878,-41.814,-179.373,5.350,148.741
C02516=1228.346,9.628,-41.800,-179.376,5.349,148.741
C02517=1228.351,9.379,-41.785,-179.378,5.349,148.742
C02518=1228.357,9.129,-41.770,-179.380,5.349,148.743
C02519=1228.361,8.880,-41.755,-179.383,5.348,148.744
C02520=1228.366,8.630,-41.740,-179.386,5.348,148.744
C02521=1228.372,8.380,-41.725,-179.388,5.348,148.745
C02522=1228.376,8.131,-41.711,-179.390,5.348,148.746
C02523=1228.381,7.882,-41.696,-179.393,5.347,148.746
C02524=1228.386,7.632,-41.681,-179.396,5.346,148.747
C02525=1228.392,7.382,-41.666,-179.398,5.347,148.748
C02526=1228.396,7.133,-41.651,-179.401,5.346,148.748
C02527=1228.401,6.883,-41.637,-179.403,5.346,148.749
C02528=1228.406,6.634,-41.622,-179.406,5.345,148.750
C02529=1228.412,6.384,-41.607,-179.408,5.345,148.750
C02530=1228.416,6.135,-41.592,-179.411,5.345,148.751
C02531=1228.421,5.885,-41.578,-179.413,5.344,148.752
C02532=1228.426,5.636,-41.564,-179.416,5.344,148.752
C02533=1228.432,5.386,-41.548,-179.418,5.344,148.753
C02534=1228.437,5.136,-41.534,-179.421,5.344,148.754
C02535=1228.442,4.887,-41.520,-179.423,5.343,148.755
C02536=1228.446,4.638,-41.505,-179.426,5.343,148.755
C02537=1228.451,4.388,-41.490,-179.428,5.343,148.756
C02538=1228.457,4.138,-41.476,-179.431,5.342,148.757
C02539=1228.462,3.869,-41.460,-179.433,5.342,148.757
C02540=1228.467,3.600,-41.444,-179.436,5.341,148.758
C02541=1228.472,3.332,-41.428,-179.439,5.341,148.759
C02542=1228.478,3.062,-41.412,-179.442,5.341,148.760
C02543=1228.483,2.813,-41.398,-179.444,5.341,148.760
C02544=1228.488,2.563,-41.384,-179.446,5.340,148.761
C02545=1228.493,2.315,-41.369,-179.449,5.340,148.762
C02546=1228.498,2.065,-41.355,-179.452,5.339,148.762
C02547=1228.503,1.815,-41.340,-179.454,5.340,148.763
C02548=1228.508,1.565,-41.326,-179.456,5.339,148.764
C02549=1228.514,1.316,-41.310,-179.459,5.339,148.764
C02550=1228.518,1.066,-41.296,-179.461,5.339,148.765
C02551=1228.523,0.817,-41.282,-179.464,5.338,148.766
C02552=1228.528,0.567,-41.268,-179.467,5.338,148.766
C02553=1228.533,0.318,-41.253,-179.469,5.337,148.767
C02554=1228.538,0.068,-41.238,-179.471,5.338,148.768
C02555=1228.544,-0.181,-41.224,-179.474,5.337,148.769
C02556=1228.549,-0.431,-41.210,-179.477,5.336,148.769
C02557=1228.553,-0.680,-41.196,-179.479,5.336,148.770
C02558=1228.558,-0.929,-41.181,-179.481,5.336,148.771
C02559=1228.564,-1.179,-41.166,-179.484,5.336,148.771
C02560=1228.569,-1.429,-41.152,-179.487,5.335,148.772
C02561=1228.574,-1.679,-41.137,-179.489,5.335,148.773
C02562=1228.579,-1.929,-41.123,-179.491,5.335,148.773
C02563=1228.584,-2.178,-41.109,-179.494,5.334,148.774
C02564=1228.589,-2.427,-41.094,-179.497,5.334,148.775
C02565=1228.594,-2.676,-41.080,-179.499,5.334,148.775
C02566=1228.599,-2.926,-41.066,-179.501,5.334,148.776
C02567=1228.604,-3.176,-41.051,-179.504,5.333,148.777
C02568=1228.609,-3.425,-41.037,-179.507,5.333,148.777
C02569=1228.614,-3.674,-41.023,-179.509,5.333,148.778
C02570=1228.619,-3.924,-41.009,-179.511,5.332,148.779
C02571=1228.624,-4.174,-40.995,-179.514,5.332,148.780
C02572=1228.629,-4.424,-40.980,-179.516,5.332,148.780
C02573=1228.634,-4.673,-40.966,-179.519,5.332,148.781
C02574=1228.639,-4.922,-40.951,-179.521,5.331,148.782
C02575=1228.644,-5.171,-40.937,-179.524,5.331,148.782
C02576=1228.649,-5.421,-40.923,-179.526,5.331,148.783
C02577=1228.654,-5.671,-40.909,-179.529,5.330,148.784
C02578=1228.659,-5.921,-40.894,-179.531,5.330,148.784
C02579=1228.664,-6.170,-40.880,-179.534,5.330,148.785
C02580=1228.670,-6.419,-40.866,-179.536,5.330,148.786
C02581=1228.675,-6.669,-40.852,-179.539,5.329,148.786
C02582=1228.680,-6.919,-40.838,-179.541,5.329,148.787
C02583=1228.685,-7.168,-40.823,-179.544,5.329,148.788
C02584=1228.689,-7.418,-40.809,-179.546,5.328,148.789
C02585=1228.694,-7.667,-40.796,-179.549,5.328,148.789
C02586=1228.699,-7.917,-40.782,-179.551,5.328,148.790
C02587=1228.704,-8.166,-40.767,-179.554,5.328,148.791
C02588=1228.709,-8.416,-40.753,-179.556,5.327,148.791
C02589=1228.715,-8.666,-40.740,-179.558,5.327,148.792
C02590=1228.720,-8.915,-40.726,-179.561,5.327,148.793
C02591=1228.725,-9.165,-40.711,-179.564,5.326,148.793
C02592=1228.730,-9.415,-40.697,-179.566,5.327,148.794
C02593=1228.735,-9.664,-40.683,-179.568,5.326,148.795
C02594=1228.740,-9.913,-40.669,-179.571,5.326,148.795
C02595=1228.745,-10.163,-40.655,-179.573,5.326,148.796
C02596=1228.750,-10.413,-40.641,-179.576,5.325,148.797
C02597=1228.755,-10.662,-40.627,-179.578,5.325,148.798
C02598=1228.760,-10.911,-40.613,-179.581,5.324,148.798
C02599=1228.765,-11.161,-40.598,-179.583,5.325,148.799
C02600=1228.770,-11.411,-40.585,-179.586,5.324,148.800
C02601=1228.776,-11.660,-40.571,-179.589,5.324,148.800
C02602=1228.780,-11.910,-40.557,-179.591,5.324,148.801
C02603=1228.785,-12.159,-40.543,-179.593,5.323,148.802
C02604=1228.790,-12.409,-40.529,-179.596,5.323,148.802
C02605=1228.796,-12.658,-40.515,-179.598,5.323,148.803
C02606=1228.801,-12.908,-40.501,-179.601,5.323,148.804
C02607=1228.805,-13.158,-40.487,-179.603,5.322,148.804
C02608=1228.811,-13.407,-40.474,-179.605,5.322,148.805
C02609=1228.816,-13.657,-40.459,-179.608,5.322,148.806
C02610=1228.820,-13.906,-40.445,-179.611,5.321,148.807
C02611=1228.826,-14.156,-40.432,-179.613,5.322,148.807
C02612=1228.831,-14.405,-40.418,-179.615,5.321,148.808
C02613=1228.836,-14.655,-40.404,-179.618,5.321,148.809
C02614=1228.841,-14.904,-40.390,-179.620,5.321,148.809
C02615=1228.846,-15.154,-40.376,-179.623,5.320,148.810
C02616=1228.851,-15.404,-40.362,-179.625,5.320,148.811
C02617=1228.856,-15.653,-40.349,-179.628,5.319,148.811
C02618=1228.861,-15.903,-40.335,-179.630,5.320,148.812
C02619=1228.866,-16.153,-40.321,-179.633,5.319,148.813
C02620=1228.872,-16.402,-40.307,-179.636,5.319,148.813
C02621=1228.876,-16.651,-40.293,-179.638,5.319,148.814
C02622=1228.881,-16.902,-40.280,-179.640,5.319,148.815
C02623=1228.887,-17.151,-40.266,-179.643,5.318,148.816
C02624=1228.891,-17.400,-40.252,-179.645,5.318,148.816
C02625=1228.896,-17.650,-40.239,-179.648,5.318,148.817
C02626=1228.902,-17.899,-40.225,-179.651,5.318,148.818
C02627=1228.907,-18.149,-40.210,-179.653,5.318,148.819
C02628=1228.912,-18.398,-40.198,-179.656,5.317,148.819
C02629=1228.917,-18.648,-40.184,-179.658,5.317,148.820
C02630=1228.922,-18.898,-40.169,-179.660,5.317,148.821
C02631=1228.927,-19.147,-40.157,-179.663,5.317,148.821
C02632=1228.932,-19.397,-40.142,-179.666,5.316,148.822
C02633=1228.937,-19.647,-40.129,-179.668,5.317,148.823
C02634=1228.942,-19.896,-40.116,-179.670,5.316,148.823
C02635=1228.947,-20.146,-40.101,-179.673,5.316,148.824
C02636=1228.953,-20.395,-40.088,-179.675,5.316,148.825
C02637=1228.957,-20.645,-40.074,-179.678,5.315,148.826
C02638=1228.962,-20.895,-40.061,-179.680,5.316,148.826
C02639=1228.968,-21.144,-40.047,-179.682,5.315,148.827
C02640=1228.972,-21.393,-40.033,-179.685,5.315,148.828
C02641=1228.978,-21.643,-40.020,-179.687,5.315,148.828
C02642=1228.983,-21.893,-40.006,-179.690,5.314,148.829
C02643=1228.988,-22.162,-39.992,-179.693,5.314,148.830
C02644=1228.994,-22.431,-39.977,-179.695,5.313,148.830
C02645=1228.999,-22.701,-39.962,-179.698,5.314,148.831
C02646=1229.005,-22.970,-39.947,-179.700,5.314,148.832
C02647=1229.010,-23.219,-39.935,-179.703,5.313,148.833
C02648=1229.015,-23.469,-39.921,-179.706,5.313,148.833
C02649=1229.019,-23.719,-39.908,-179.708,5.313,148.834
C02650=1229.025,-23.968,-39.894,-179.711,5.312,148.835
C02651=1229.030,-24.218,-39.880,-179.713,5.313,148.835
C02652=1229.035,-24.467,-39.867,-179.715,5.312,148.836
C02653=1229.040,-24.717,-39.853,-179.718,5.312,148.837
C02654=1229.045,-24.966,-39.840,-179.720,5.312,148.838
C02655=1229.050,-25.216,-39.826,-179.723,5.311,148.838
C02656=1229.055,-25.465,-39.813,-179.725,5.311,148.839
C02657=1229.061,-25.715,-39.800,-179.727,5.311,148.840
C02658=1229.066,-25.965,-39.787,-179.730,5.311,148.840
C02659=1229.071,-26.214,-39.773,-179.733,5.310,148.841
C02660=1229.076,-26.464,-39.760,-179.735,5.311,148.842
C02661=1229.081,-26.713,-39.746,-179.737,5.310,148.842
C02662=1229.086,-26.963,-39.733,-179.740,5.310,148.843
C02663=1229.091,-27.213,-39.720,-179.742,5.310,148.844
C02664=1229.096,-27.462,-39.706,-179.745,5.309,148.845
C02665=1229.101,-27.712,-39.693,-179.747,5.310,148.845
C02666=1229.106,-27.961,-39.680,-179.750,5.310,148.846
C02667=1229.111,-28.211,-39.666,-179.753,5.309,148.847
C02668=1229.116,-28.460,-39.653,-179.755,5.309,148.848
C02669=1229.121,-28.710,-39.639,-179.758,5.309,148.848
C02670=1229.126,-28.959,-39.626,-179.760,5.308,148.849
C02671=1229.132,-29.210,-39.613,-179.762,5.309,148.850
C02672=1229.137,-29.459,-39.600,-179.765,5.308,148.850
C02673=1229.142,-29.709,-39.586,-179.768,5.308,148.851
C02674=1229.147,-29.958,-39.573,-179.770,5.308,148.852
C02675=1229.152,-30.209,-39.560,-179.772,5.307,148.852
C02676=1229.157,-30.457,-39.546,-179.774,5.308,148.853
C02677=1229.161,-30.707,-39.534,-179.777,5.307,148.854
C02678=1229.167,-30.957,-39.520,-179.780,5.307,148.855
C02679=1229.172,-31.206,-39.507,-179.782,5.307,148.855
C02680=1229.177,-31.456,-39.493,-179.784,5.307,148.856
C02681=1229.183,-31.705,-39.481,-179.787,5.306,148.857
C02682=1229.188,-31.956,-39.467,-179.789,5.306,148.857
C02683=1229.193,-32.204,-39.454,-179.792,5.306,148.858
C02684=1229.197,-32.454,-39.441,-179.794,5.306,148.859
C02685=1229.203,-32.704,-39.428,-179.797,5.306,148.859
C02686=1229.208,-32.954,-39.415,-179.799,5.305,148.860
C02687=1229.213,-33.204,-39.402,-179.801,5.306,148.861
C02688=1229.218,-33.452,-39.388,-179.804,5.305,148.862
C02689=1229.223,-33.702,-39.375,-179.807,5.305,148.862
C02690=1229.229,-33.952,-39.362,-179.809,5.305,148.863
C02691=1229.233,-34.202,-39.349,-179.811,5.304,148.864
C02692=1229.238,-34.451,-39.337,-179.814,5.305,148.864
C02693=1229.244,-34.701,-39.323,-179.816,5.304,148.865
C02694=1229.248,-34.950,-39.310,-179.819,5.304,148.866
C02695=1229.253,-35.200,-39.297,-179.821,5.304,148.866
C02696=1229.259,-35.450,-39.284,-179.824,5.304,148.867
C02697=1229.264,-35.699,-39.271,-179.826,5.304,148.868
C02698=1229.269,-35.949,-39.258,-179.829,5.304,148.869
C02699=1229.274,-36.199,-39.245,-179.831,5.303,148.869
C02700=1229.279,-36.448,-39.232,-179.834,5.304,148.870
C02701=1229.284,-36.697,-39.220,-179.836,5.303,148.871
C02702=1229.289,-36.947,-39.205,-179.839,5.303,148.872
C02703=1229.295,-37.197,-39.193,-179.841,5.303,148.872
C02704=1229.300,-37.446,-39.180,-179.844,5.302,148.873
C02705=1229.305,-37.696,-39.167,-179.846,5.303,148.874
C02706=1229.310,-37.945,-39.154,-179.848,5.302,148.874
C02707=1229.315,-38.195,-39.141,-179.851,5.302,148.875
C02708=1229.320,-38.445,-39.128,-179.853,5.302,148.876
C02709=1229.326,-38.694,-39.115,-179.856,5.302,148.876
C02710=1229.330,-38.944,-39.102,-179.858,5.302,148.877
C02711=1229.335,-39.194,-39.090,-179.861,5.301,148.878
C02712=1229.341,-39.443,-39.076,-179.863,5.301,148.879
C02713=1229.346,-39.693,-39.063,-179.865,5.301,148.879
C02714=1229.351,-39.943,-39.051,-179.868,5.301,148.880
C02715=1229.356,-40.192,-39.038,-179.870,5.301,148.881
C02716=1229.362,-40.442,-39.025,-179.873,5.300,148.881
C02717=1229.366,-40.692,-39.012,-179.875,5.300,148.882
C02718=1229.371,-40.941,-38.999,-179.877,5.300,148.883
C02719=1229.376,-41.190,-38.987,-179.880,5.300,148.883
C02720=1229.381,-41.440,-38.974,-179.882,5.300,148.884
C02721=1229.387,-41.690,-38.961,-179.885,5.300,148.885
C02722=1229.392,-41.939,-38.948,-179.888,5.299,148.886
C02723=1229.397,-42.189,-38.935,-179.890,5.299,148.886
C02724=1229.402,-42.439,-38.923,-179.892,5.299,148.887
C02725=1229.407,-42.688,-38.910,-179.894,5.299,148.888
C02726=1229.413,-42.938,-38.897,-179.897,5.299,148.888
C02727=1229.417,-43.188,-38.884,-179.900,5.298,148.889
C02728=1229.423,-43.438,-38.872,-179.902,5.299,148.890
C02729=1229.428,-43.687,-38.859,-179.904,5.298,148.890
C02730=1229.432,-43.937,-38.846,-179.907,5.299,148.891
C02731=1229.437,-44.186,-38.834,-179.910,5.298,148.892
C02732=1229.442,-44.436,-38.821,-179.912,5.299,148.893
C02733=1229.448,-44.685,-38.808,-179.914,5.298,148.894
C02734=1229.453,-44.935,-38.795,-179.917,5.298,148.894
C02735=1229.458,-45.184,-38.782,-179.919,5.298,148.895
C02736=1229.463,-45.434,-38.770,-179.922,5.298,148.896
C02737=1229.469,-45.684,-38.758,-179.924,5.298,148.896
C02738=1229.473,-45.934,-38.745,-179.927,5.297,148.897
C02739=1229.478,-46.183,-38.732,-179.929,5.297,148.898
C02740=1229.484,-46.433,-38.719,-179.931,5.297,148.898
C02741=1229.489,-46.682,-38.707,-179.934,5.297,148.899
C02742=1229.494,-46.933,-38.694,-179.936,5.297,148.900
C02743=1229.499,-47.182,-38.682,-179.939,5.297,148.901
C02744=1229.504,-47.431,-38.669,-179.941,5.297,148.901
C02745=1229.509,-47.681,-38.656,-179.944,5.296,148.902
C02746=1229.514,-47.930,-38.644,-179.946,5.296,148.903
C02747=1229.520,-48.200,-38.631,-179.948,5.296,148.903
C02748=1229.526,-48.470,-38.617,-179.951,5.296,148.904
C02749=1229.531,-48.739,-38.603,-179.954,5.296,148.905
C02750=1229.536,-49.010,-38.590,-179.956,5.296,148.906
C02751=1229.542,-49.259,-38.578,-179.959,5.296,148.906
C02752=1229.547,-49.508,-38.565,-179.962,5.295,148.907
C02753=1229.551,-49.758,-38.552,-179.964,5.295,148.908
C02754=1229.557,-50.009,-38.540,-179.966,5.295,148.908
C02755=1229.562,-50.258,-38.527,-179.968,5.295,148.909
C02756=1229.568,-50.507,-38.514,-179.971,5.295,148.910
C02757=1229.573,-50.757,-38.503,-179.973,5.295,148.911
C02758=1229.578,-51.007,-38.490,-179.976,5.295,148.911
C02759=1229.583,-51.256,-38.477,-179.978,5.294,148.912
C02760=1229.588,-51.506,-38.465,-179.981,5.294,148.913
C02761=1229.593,-51.756,-38.453,-179.983,5.294,148.913
C02762=1229.598,-52.005,-38.440,-179.985,5.294,148.914
C02763=1229.604,-52.255,-38.428,-179.988,5.294,148.915
C02764=1229.608,-52.505,-38.415,-179.990,5.294,148.916
C02765=1229.613,-52.754,-38.402,-179.993,5.294,148.916
C02766=1229.618,-53.004,-38.391,-179.995,5.293,148.917
C02767=1229.623,-53.253,-38.379,-179.997,5.293,148.918
C02768=1229.628,-53.503,-38.366,179.999,5.293,148.919
C02769=1229.634,-53.753,-38.354,179.997,5.294,148.919
C02770=1229.639,-54.002,-38.342,179.995,5.293,148.920
C02771=1229.644,-54.252,-38.329,179.993,5.294,148.921
C02772=1229.649,-54.502,-38.317,179.990,5.293,148.921
C02773=1229.654,-54.751,-38.304,179.987,5.293,148.922
C02774=1229.659,-55.001,-38.292,179.985,5.293,148.923
C02775=1229.665,-55.250,-38.280,179.982,5.292,148.924
C02776=1229.670,-55.500,-38.268,179.980,5.293,148.924
C02777=1229.675,-55.750,-38.255,179.978,5.292,148.925
C02778=1229.681,-56.000,-38.243,179.976,5.293,148.926
C02779=1229.685,-56.250,-38.230,179.973,5.292,148.926
C02780=1229.690,-56.499,-38.219,179.971,5.292,148.927
C02781=1229.695,-56.749,-38.206,179.968,5.292,148.928
C02782=1229.700,-56.998,-38.194,179.966,5.292,148.928
C02783=1229.705,-57.248,-38.182,179.963,5.292,148.929
C02784=1229.711,-57.498,-38.170,179.961,5.291,148.930
C02785=1229.716,-57.747,-38.157,179.959,5.292,148.931
C02786=1229.721,-57.997,-38.145,179.956,5.291,148.931
C02787=1229.727,-58.246,-38.133,179.954,5.292,148.932
C02788=1229.731,-58.496,-38.122,179.951,5.291,148.933
C02789=1229.736,-58.745,-38.109,179.949,5.291,148.933
C02790=1229.742,-58.995,-38.097,179.947,5.291,148.934
C02791=1229.746,-59.245,-38.084,179.944,5.290,148.935
C02792=1229.752,-59.495,-38.072,179.942,5.291,148.935
C02793=1229.757,-59.744,-38.060,179.939,5.290,148.936
C02794=1229.762,-59.994,-38.048,179.937,5.291,148.937
C02795=1229.767,-60.244,-38.036,179.934,5.290,148.938
C02796=1229.772,-60.493,-38.024,179.932,5.291,148.938
C02797=1229.778,-60.743,-38.012,179.930,5.290,148.939
C02798=1229.783,-60.993,-37.999,179.927,5.290,148.940
C02799=1229.787,-61.242,-37.988,179.925,5.290,148.940
C02800=1229.793,-61.492,-37.976,179.922,5.289,148.941
C02801=1229.798,-61.741,-37.964,179.920,5.290,148.942
C02802=1229.803,-61.991,-37.952,179.917,5.289,148.943
C02803=1229.808,-62.241,-37.939,179.915,5.290,148.943
C02804=1229.813,-62.490,-37.928,179.913,5.289,148.944
C02805=1229.819,-62.740,-37.916,179.911,5.289,148.945
C02806=1229.824,-62.990,-37.903,179.908,5.289,148.945
C02807=1229.829,-63.240,-37.891,179.906,5.289,148.946
C02808=1229.834,-63.489,-37.880,179.903,5.289,148.947
C02809=1229.839,-63.738,-37.868,179.901,5.289,148.947
C02810=1229.844,-63.988,-37.856,179.898,5.289,148.948
C02811=1229.850,-64.238,-37.844,179.896,5.288,148.949
C02812=1229.854,-64.487,-37.832,179.894,5.289,148.950
C02813=1229.860,-64.737,-37.820,179.891,5.288,148.950
C02814=1229.865,-64.987,-37.808,179.889,5.288,148.951
C02815=1229.870,-65.237,-37.796,179.886,5.288,148.952
C02816=1229.875,-65.486,-37.784,179.884,5.288,148.952
C02817=1229.880,-65.736,-37.772,179.881,5.288,148.953
C02818=1229.886,-65.986,-37.760,179.879,5.288,148.954
C02819=1229.890,-66.236,-37.749,179.877,5.288,148.955
C02820=1229.896,-66.485,-37.736,179.875,5.288,148.955
C02821=1229.901,-66.735,-37.725,179.871,5.288,148.956
C02822=1229.906,-66.985,-37.713,179.869,5.288,148.957
C02823=1229.911,-67.234,-37.701,179.867,5.288,148.958
C02824=1229.916,-67.484,-37.689,179.864,5.287,148.958
C02825=1229.921,-67.733,-37.678,179.862,5.288,148.959
C02826=1229.926,-67.983,-37.666,179.859,5.287,148.960
C02827=1229.932,-68.233,-37.654,179.857,5.288,148.960
C02828=1229.937,-68.482,-37.643,179.854,5.287,148.961
C02829=1229.942,-68.732,-37.630,179.852,5.287,148.962
C02830=1229.948,-68.981,-37.618,179.850,5.287,148.963
C02831=1229.952,-69.231,-37.607,179.848,5.287,148.963
C02832=1229.958,-69.481,-37.595,179.845,5.287,148.964
C02833=1229.963,-69.731,-37.583,179.843,5.287,148.965
C02834=1229.968,-69.981,-37.572,179.840,5.287,148.965
C02835=1229.973,-70.231,-37.560,179.838,5.287,148.966
C02836=1229.978,-70.480,-37.548,179.835,5.287,148.967
C02837=1229.983,-70.729,-37.536,179.833,5.287,148.967
C02838=1229.989,-70.979,-37.524,179.831,5.286,148.968
C02839=1229.994,-71.228,-37.513,179.829,5.287,148.969
C02840=1229.999,-71.478,-37.502,179.826,5.286,148.970
C02841=1230.005,-71.728,-37.490,179.824,5.287,148.970
C02842=1230.009,-71.978,-37.478,179.821,5.286,148.971
C02843=1230.015,-72.228,-37.466,179.818,5.286,148.972
C02844=1230.020,-72.477,-37.455,179.816,5.286,148.972
C02845=1230.025,-72.727,-37.443,179.814,5.286,148.973
C02846=1230.029,-72.976,-37.431,179.812,5.286,148.974
C02847=1230.035,-73.226,-37.420,179.809,5.286,148.975
C02848=1230.041,-73.476,-37.408,179.807,5.286,148.975
C02849=1230.045,-73.725,-37.397,179.804,5.285,148.976
C02850=1230.051,-73.975,-37.385,179.802,5.286,148.977
C02851=1230.057,-74.246,-37.372,179.799,5.285,148.977
C02852=1230.062,-74.516,-37.360,179.797,5.286,148.978
C02853=1230.068,-74.786,-37.347,179.795,5.285,148.979
C02854=1230.073,-75.057,-37.335,179.792,5.285,148.980
C02855=1230.079,-75.306,-37.324,179.789,5.285,148.980
C02856=1230.084,-75.556,-37.312,179.787,5.285,148.981
C02857=1230.089,-75.806,-37.301,179.785,5.285,148.982
C02858=1230.094,-76.055,-37.289,179.782,5.285,148.983
C02859=1230.099,-76.305,-37.277,179.780,5.285,148.983
C02860=1230.104,-76.555,-37.265,179.777,5.285,148.984
C02861=1230.110,-76.804,-37.255,179.775,5.285,148.985
C02862=1230.115,-77.054,-37.243,179.772,5.285,148.985
C02863=1230.120,-77.304,-37.231,179.770,5.285,148.986
C02864=1230.124,-77.553,-37.220,179.768,5.285,148.987
C02865=1230.130,-77.803,-37.208,179.766,5.285,148.988
C02866=1230.135,-78.052,-37.197,179.763,5.284,148.988
C02867=1230.141,-78.303,-37.186,179.761,5.285,148.989
C02868=1230.146,-78.552,-37.175,179.758,5.284,148.990
C02869=1230.151,-78.802,-37.163,179.756,5.285,148.990
C02870=1230.156,-79.052,-37.152,179.753,5.284,148.991
C02871=1230.162,-79.301,-37.140,179.751,5.285,148.992
C02872=1230.166,-79.551,-37.129,179.749,5.284,148.993
C02873=1230.171,-79.800,-37.118,179.746,5.284,148.993
C02874=1230.177,-80.050,-37.106,179.744,5.284,148.994
C02875=1230.181,-80.300,-37.094,179.741,5.283,148.995
C02876=1230.188,-80.550,-37.084,179.739,5.284,148.995
C02877=1230.192,-80.799,-37.072,179.736,5.283,148.996
C02878=1230.198,-81.049,-37.060,179.734,5.284,148.997
C02879=1230.202,-81.299,-37.049,179.732,5.283,148.998
C02880=1230.208,-81.548,-37.038,179.730,5.284,148.998
C02881=1230.213,-81.798,-37.026,179.727,5.283,148.999
C02882=1230.218,-82.048,-37.016,179.725,5.283,148.999
C02883=1230.223,-82.298,-37.004,179.723,5.283,149.000
C02884=1230.229,-82.547,-36.993,179.721,5.283,149.001
C02885=1230.234,-82.796,-36.982,179.718,5.283,149.002
C02886=1230.239,-83.047,-36.970,179.716,5.283,149.002
C02887=1230.244,-83.297,-36.959,179.713,5.282,149.003
C02888=1230.249,-83.546,-36.948,179.711,5.283,149.004
C02889=1230.255,-83.795,-36.936,179.708,5.282,149.004
C02890=1230.259,-84.045,-36.925,179.706,5.283,149.005
C02891=1230.264,-84.295,-36.914,179.704,5.282,149.006
C02892=1230.270,-84.545,-36.903,179.702,5.283,149.006
C02893=1230.275,-84.794,-36.892,179.699,5.282,149.007
C02894=1230.280,-85.044,-36.881,179.697,5.282,149.008
C02895=1230.286,-85.294,-36.870,179.694,5.282,149.009
C02896=1230.291,-85.543,-36.858,179.692,5.282,149.009
C02897=1230.295,-85.793,-36.847,179.689,5.282,149.010
C02898=1230.300,-86.043,-36.836,179.687,5.282,149.011
C02899=1230.307,-86.292,-36.825,179.685,5.282,149.011
C02900=1230.311,-86.542,-36.814,179.682,5.282,149.012
C02901=1230.316,-86.792,-36.803,179.680,5.282,149.013
C02902=1230.322,-87.042,-36.792,179.678,5.282,149.014
C02903=1230.327,-87.291,-36.780,179.675,5.282,149.014
C02904=1230.332,-87.541,-36.770,179.673,5.282,149.015
C02905=1230.337,-87.790,-36.759,179.670,5.282,149.016
C02906=1230.343,-88.040,-36.747,179.668,5.282,149.016
C02907=1230.348,-88.291,-36.736,179.665,5.281,149.017
C02908=1230.353,-88.539,-36.725,179.663,5.282,149.018
C02909=1230.358,-88.789,-36.714,179.661,5.281,149.019
C02910=1230.363,-89.040,-36.703,179.659,5.282,149.019
C02911=1230.369,-89.289,-36.692,179.657,5.282,149.020
C02912=1230.374,-89.539,-36.681,179.654,5.282,149.021
C02913=1230.378,-89.788,-36.670,179.652,5.282,149.021
C02914=1230.384,-90.038,-36.659,179.649,5.281,149.022
C02915=1230.389,-90.288,-36.648,179.647,5.282,149.023
C02916=1230.394,-90.538,-36.637,179.644,5.281,149.024
C02917=1230.400,-90.787,-36.627,179.642,5.282,149.024
C02918=1230.404,-91.037,-36.615,179.640,5.281,149.025
C02919=1230.410,-91.287,-36.604,179.637,5.282,149.026
C02920=1230.415,-91.536,-36.593,179.635,5.281,149.026
C02921=1230.420,-91.786,-36.583,179.633,5.282,149.027
C02922=1230.426,-92.035,-36.572,179.630,5.281,149.028
C02923=1230.430,-92.285,-36.560,179.628,5.281,149.028
C02924=1230.435,-92.535,-36.550,179.626,5.281,149.029
C02925=1230.441,-92.784,-36.538,179.624,5.281,149.030
C02926=1230.446,-93.035,-36.528,179.621,5.281,149.030
C02927=1230.452,-93.284,-36.517,179.619,5.281,149.031
C02928=1230.457,-93.534,-36.506,179.616,5.280,149.032
C02929=1230.461,-93.783,-36.495,179.614,5.281,149.033
C02930=1230.467,-94.033,-36.485,179.611,5.280,149.033
C02931=1230.473,-94.284,-36.474,179.609,5.281,149.034
C02932=1230.478,-94.532,-36.463,179.607,5.280,149.035
C02933=1230.483,-94.783,-36.452,179.605,5.281,149.035
C02934=1230.488,-95.032,-36.441,179.602,5.280,149.036
C02935=1230.493,-95.282,-36.431,179.600,5.281,149.037
C02936=1230.498,-95.532,-36.419,179.597,5.280,149.038
C02937=1230.504,-95.781,-36.409,179.595,5.280,149.038
C02938=1230.508,-96.031,-36.398,179.592,5.280,149.039
C02939=1230.515,-96.281,-36.387,179.590,5.280,149.040
C02940=1230.520,-96.531,-36.376,179.588,5.280,149.040
C02941=1230.524,-96.780,-36.365,179.586,5.280,149.041
C02942=1230.530,-97.030,-36.355,179.583,5.280,149.042
C02943=1230.535,-97.280,-36.344,179.581,5.280,149.043
C02944=1230.540,-97.529,-36.333,179.579,5.281,149.043
C02945=1230.545,-97.779,-36.323,179.576,5.280,149.044
C02946=1230.550,-98.028,-36.312,179.574,5.280,149.044
C02947=1230.555,-98.279,-36.301,179.572,5.280,149.045
C02948=1230.561,-98.528,-36.291,179.570,5.280,149.046
C02949=1230.566,-98.778,-36.280,179.567,5.280,149.047
C02950=1230.571,-99.027,-36.270,179.565,5.280,149.047
C02951=1230.576,-99.278,-36.259,179.562,5.279,149.048
C02952=1230.582,-99.526,-36.248,179.560,5.280,149.049
C02953=1230.587,-99.777,-36.237,179.557,5.279,149.049
C02954=1230.592,-100.027,-36.227,179.555,5.280,149.050
C02955=1230.598,-100.297,-36.215,179.553,5.279,149.051
C02956=1230.604,-100.569,-36.203,179.551,5.280,149.052
C02957=1230.609,-100.839,-36.192,179.547,5.280,149.053
C02958=1230.615,-101.110,-36.181,179.545,5.279,149.053
C02959=1230.620,-101.360,-36.169,179.543,5.280,149.054
C02960=1230.625,-101.610,-36.159,179.540,5.279,149.055
C02961=1230.630,-101.860,-36.149,179.538,5.279,149.055
C02962=1230.636,-102.109,-36.138,179.536,5.280,149.056
C02963=1230.641,-102.359,-36.127,179.533,5.279,149.057
C02964=1230.646,-102.608,-36.117,179.531,5.279,149.057
C02965=1230.651,-102.859,-36.106,179.529,5.279,149.058
C02966=1230.657,-103.108,-36.096,179.527,5.279,149.059
C02967=1230.661,-103.358,-36.085,179.524,5.279,149.059
C02968=1230.667,-103.607,-36.075,179.522,5.279,149.060
C02969=1230.672,-103.857,-36.065,179.519,5.279,149.061
C02970=1230.677,-104.107,-36.054,179.517,5.279,149.062
C02971=1230.682,-104.357,-36.044,179.515,5.279,149.062
C02972=1230.687,-104.606,-36.033,179.512,5.279,149.063
C02973=1230.693,-104.856,-36.023,179.510,5.279,149.064
C02974=1230.698,-105.106,-36.012,179.508,5.279,149.064
C02975=1230.704,-105.355,-36.002,179.505,5.279,149.065
C02976=1230.709,-105.606,-35.991,179.503,5.279,149.066
C02977=1230.714,-105.855,-35.981,179.500,5.278,149.067
C02978=1230.719,-106.105,-35.970,179.498,5.279,149.067
C02979=1230.724,-106.354,-35.960,179.497,5.279,149.068
C02980=1230.729,-106.604,-35.950,179.494,5.278,149.069
C02981=1230.734,-106.854,-35.939,179.492,5.279,149.069
C02982=1230.740,-107.103,-35.929,179.489,5.278,149.070
C02983=1230.745,-107.354,-35.919,179.487,5.279,149.071
C02984=1230.751,-107.603,-35.908,179.484,5.278,149.071
C02985=1230.756,-107.853,-35.898,179.482,5.279,149.072
C02986=1230.761,-108.102,-35.887,179.480,5.278,149.073
C02987=1230.766,-108.352,-35.877,179.477,5.279,149.074
C02988=1230.771,-108.602,-35.867,179.475,5.278,149.074
C02989=1230.776,-108.851,-35.857,179.473,5.278,149.075
C02990=1230.781,-109.102,-35.846,179.470,5.278,149.076
C02991=1230.787,-109.351,-35.836,179.468,5.278,149.076
C02992=1230.792,-109.601,-35.826,179.466,5.278,149.077
C02993=1230.797,-109.851,-35.815,179.464,5.278,149.078
C02994=1230.803,-110.101,-35.805,179.462,5.278,149.078
C02995=1230.807,-110.350,-35.795,179.459,5.278,149.079
C02996=1230.813,-110.600,-35.785,179.457,5.278,149.080
C02997=1230.819,-110.850,-35.774,179.454,5.278,149.080
C02998=1230.824,-111.100,-35.764,179.452,5.278,149.081
C02999=1230.829,-111.349,-35.754,179.449,5.278,149.082
C03000=1230.834,-111.599,-35.744,179.447,5.278,149.083
C03001=1230.839,-111.849,-35.733,179.445,5.278,149.083
C03002=1230.845,-112.098,-35.723,179.443,5.278,149.084
C03003=1230.850,-112.348,-35.713,179.440,5.277,149.084
C03004=1230.855,-112.598,-35.702,179.438,5.278,149.085
C03005=1230.860,-112.847,-35.693,179.436,5.278,149.086
C03006=1230.866,-113.097,-35.683,179.433,5.278,149.087
C03007=1230.871,-113.347,-35.672,179.431,5.278,149.087
C03008=1230.876,-113.597,-35.662,179.429,5.278,149.088
C03009=1230.881,-113.846,-35.652,179.427,5.278,149.089
C03010=1230.886,-114.096,-35.642,179.424,5.277,149.089
C03011=1230.892,-114.346,-35.631,179.422,5.278,149.090
C03012=1230.897,-114.595,-35.621,179.419,5.277,149.091
C03013=1230.902,-114.845,-35.611,179.417,5.277,149.091
C03014=1230.907,-115.095,-35.602,179.415,5.277,149.092
C03015=1230.913,-115.345,-35.592,179.413,5.277,149.093
C03016=1230.918,-115.595,-35.581,179.411,5.278,149.094
C03017=1230.923,-115.844,-35.571,179.408,5.277,149.094
C03018=1230.928,-116.094,-35.561,179.406,5.278,149.095
C03019=1230.933,-116.344,-35.551,179.403,5.277,149.096
C03020=1230.938,-116.593,-35.541,179.401,5.278,149.096
C03021=1230.944,-116.843,-35.531,179.398,5.277,149.097
C03022=1230.949,-117.094,-35.521,179.397,5.277,149.098
C03023=1230.955,-117.343,-35.511,179.394,5.277,149.098
C03024=1230.960,-117.593,-35.501,179.392,5.277,149.099
C03025=1230.965,-117.842,-35.491,179.390,5.277,149.100
C03026=1230.970,-118.092,-35.480,179.387,5.277,149.100
C03027=1230.975,-118.342,-35.471,179.385,5.277,149.101
C03028=1230.981,-118.592,-35.461,179.382,5.277,149.102
C03029=1230.986,-118.842,-35.451,179.380,5.277,149.103
C03030=1230.991,-119.091,-35.441,179.378,5.277,149.103
C03031=1230.997,-119.341,-35.431,179.376,5.277,149.104
C03032=1231.001,-119.590,-35.421,179.373,5.276,149.105
C03033=1231.007,-119.841,-35.411,179.371,5.277,149.105
C03034=1231.012,-120.090,-35.401,179.369,5.276,149.106
C03035=1231.017,-120.340,-35.391,179.367,5.277,149.107
C03036=1231.023,-120.589,-35.381,179.364,5.277,149.107
C03037=1231.028,-120.840,-35.371,179.362,5.277,149.108
C03038=1231.033,-121.089,-35.362,179.360,5.277,149.109
C03039=1231.039,-121.339,-35.352,179.357,5.276,149.109
C03040=1231.043,-121.588,-35.342,179.355,5.277,149.110
C03041=1231.049,-121.839,-35.332,179.353,5.276,149.111
C03042=1231.054,-122.088,-35.322,179.351,5.277,149.111
C03043=1231.059,-122.338,-35.312,179.348,5.276,149.112
C03044=1231.065,-122.587,-35.302,179.346,5.277,149.113
C03045=1231.070,-122.837,-35.293,179.344,5.277,149.114
C03046=1231.075,-123.087,-35.283,179.341,5.277,149.114
C03047=1231.080,-123.337,-35.272,179.339,5.277,149.115
C03048=1231.086,-123.587,-35.264,179.337,5.276,149.116
C03049=1231.091,-123.836,-35.253,179.335,5.276,149.116
C03050=1231.096,-124.086,-35.244,179.332,5.276,149.117
C03051=1231.101,-124.336,-35.234,179.330,5.276,149.118
C03052=1231.106,-124.586,-35.224,179.327,5.276,149.118
C03053=1231.112,-124.835,-35.214,179.325,5.276,149.119
C03054=1231.117,-125.085,-35.205,179.324,5.276,149.120
C03055=1231.123,-125.335,-35.195,179.321,5.276,149.120
C03056=1231.127,-125.584,-35.185,179.319,5.276,149.121
C03057=1231.133,-125.835,-35.175,179.316,5.276,149.122
C03058=1231.138,-126.084,-35.165,179.314,5.276,149.123
C03059=1230.717,-126.095,-35.202,179.310,5.279,149.124
C03060=1230.711,-125.845,-35.210,179.312,5.279,149.124
C03061=1230.706,-125.596,-35.221,179.314,5.280,149.123
C03062=1230.700,-125.346,-35.231,179.316,5.280,149.122
C03063=1230.696,-125.095,-35.240,179.318,5.279,149.122
C03064=1230.690,-124.846,-35.250,179.321,5.280,149.121
C03065=1230.685,-124.596,-35.259,179.323,5.279,149.120
C03066=1230.679,-124.346,-35.269,179.326,5.280,149.120
C03067=1230.675,-124.097,-35.279,179.327,5.280,149.119
C03068=1230.669,-123.846,-35.289,179.330,5.280,149.118
C03069=1230.664,-123.597,-35.299,179.332,5.280,149.118
C03070=1230.659,-123.348,-35.309,179.335,5.280,149.117
C03071=1230.654,-123.098,-35.318,179.337,5.280,149.116
C03072=1230.648,-122.848,-35.328,179.339,5.279,149.116
C03073=1230.643,-122.598,-35.338,179.342,5.280,149.115
C03074=1230.638,-122.349,-35.348,179.343,5.280,149.114
C03075=1230.632,-122.099,-35.358,179.346,5.280,149.114
C03076=1230.627,-121.849,-35.367,179.348,5.280,149.113
C03077=1230.622,-121.600,-35.377,179.351,5.280,149.112
C03078=1230.616,-121.349,-35.387,179.353,5.280,149.111
C03079=1230.612,-121.100,-35.397,179.356,5.280,149.111
C03080=1230.606,-120.850,-35.407,179.358,5.280,149.110
C03081=1230.601,-120.601,-35.417,179.360,5.281,149.110
C03082=1230.596,-120.350,-35.427,179.362,5.280,149.109
C03083=1230.590,-120.101,-35.437,179.364,5.280,149.108
C03084=1230.585,-119.851,-35.446,179.367,5.280,149.107
C03085=1230.580,-119.602,-35.457,179.369,5.280,149.107
C03086=1230.574,-119.351,-35.466,179.372,5.280,149.106
C03087=1230.570,-119.102,-35.476,179.374,5.280,149.105
C03088=1230.564,-118.852,-35.486,179.376,5.280,149.105
C03089=1230.558,-118.603,-35.496,179.378,5.280,149.104
C03090=1230.554,-118.353,-35.506,179.381,5.281,149.103
C03091=1230.548,-118.102,-35.516,179.383,5.281,149.103
C03092=1230.543,-117.853,-35.526,179.385,5.280,149.102
C03093=1230.538,-117.603,-35.536,179.388,5.281,149.101
C03094=1230.533,-117.353,-35.546,179.390,5.280,149.100
C03095=1230.527,-117.104,-35.557,179.392,5.281,149.100
C03096=1230.522,-116.855,-35.566,179.394,5.280,149.099
C03097=1230.517,-116.604,-35.576,179.397,5.281,149.098
C03098=1230.511,-116.354,-35.586,179.399,5.281,149.098
C03099=1230.507,-116.105,-35.596,179.401,5.281,149.097
C03100=1230.502,-115.855,-35.606,179.403,5.281,149.096
C03101=1230.496,-115.605,-35.617,179.406,5.281,149.096
C03102=1230.491,-115.356,-35.626,179.408,5.281,149.095
C03103=1230.486,-115.106,-35.637,179.410,5.280,149.094
C03104=1230.481,-114.856,-35.647,179.413,5.281,149.094
C03105=1230.475,-114.607,-35.657,179.415,5.281,149.093
C03106=1230.470,-114.356,-35.666,179.418,5.281,149.092
C03107=1230.465,-114.107,-35.677,179.419,5.281,149.092
C03108=1230.459,-113.857,-35.687,179.422,5.281,149.091
C03109=1230.454,-113.608,-35.697,179.424,5.281,149.090
C03110=1230.449,-113.358,-35.707,179.427,5.281,149.089
C03111=1230.444,-113.108,-35.717,179.429,5.281,149.089
C03112=1230.438,-112.858,-35.728,179.432,5.282,149.088
C03113=1230.433,-112.608,-35.738,179.434,5.281,149.087
C03114=1230.428,-112.359,-35.748,179.436,5.281,149.087
C03115=1230.423,-112.109,-35.758,179.438,5.281,149.086
C03116=1230.418,-111.859,-35.768,179.441,5.281,149.085
C03117=1230.412,-111.610,-35.779,179.443,5.281,149.084
C03118=1230.407,-111.359,-35.789,179.445,5.281,149.084
C03119=1230.402,-111.110,-35.799,179.447,5.282,149.083
C03120=1230.397,-110.861,-35.809,179.450,5.281,149.083
C03121=1230.392,-110.610,-35.820,179.452,5.282,149.082
C03122=1230.386,-110.361,-35.830,179.454,5.281,149.081
C03123=1230.380,-110.111,-35.840,179.457,5.282,149.080
C03124=1230.375,-109.861,-35.851,179.459,5.281,149.080
C03125=1230.371,-109.612,-35.860,179.461,5.281,149.079
C03126=1230.366,-109.362,-35.871,179.464,5.282,149.078
C03127=1230.360,-109.112,-35.881,179.466,5.281,149.078
C03128=1230.354,-108.863,-35.891,179.469,5.282,149.077
C03129=1230.349,-108.612,-35.902,179.470,5.282,149.076
C03130=1230.344,-108.363,-35.912,179.473,5.282,149.076
C03131=1230.339,-108.113,-35.922,179.475,5.282,149.075
C03132=1230.334,-107.864,-35.933,179.478,5.282,149.074
C03133=1230.329,-107.614,-35.943,179.480,5.282,149.073
C03134=1230.324,-107.364,-35.954,179.482,5.282,149.073
C03135=1230.318,-107.115,-35.964,179.485,5.282,149.072
C03136=1230.313,-106.864,-35.975,179.487,5.282,149.071
C03137=1230.307,-106.615,-35.985,179.489,5.282,149.071
C03138=1230.302,-106.365,-35.995,179.492,5.282,149.070
C03139=1230.298,-106.115,-36.005,179.494,5.282,149.069
C03140=1230.292,-105.866,-36.015,179.496,5.282,149.068
C03141=1230.287,-105.616,-36.026,179.498,5.282,149.068
C03142=1230.282,-105.367,-36.037,179.500,5.282,149.067
C03143=1230.277,-105.116,-36.047,179.503,5.283,149.067
C03144=1230.271,-104.867,-36.057,179.505,5.282,149.066
C03145=1230.266,-104.617,-36.068,179.508,5.283,149.065
C03146=1230.260,-104.367,-36.078,179.510,5.282,149.064
C03147=1230.255,-104.118,-36.089,179.513,5.283,149.064
C03148=1230.250,-103.868,-36.100,179.515,5.282,149.063
C03149=1230.245,-103.618,-36.110,179.517,5.283,149.062
C03150=1230.240,-103.368,-36.120,179.520,5.282,149.062
C03151=1230.234,-103.119,-36.131,179.522,5.283,149.061
C03152=1230.229,-102.869,-36.142,179.524,5.282,149.060
C03153=1230.224,-102.620,-36.152,179.527,5.283,149.059
C03154=1230.219,-102.369,-36.162,179.529,5.283,149.059
C03155=1230.214,-102.120,-36.172,179.531,5.283,149.058
C03156=1230.209,-101.870,-36.184,179.533,5.283,149.058
C03157=1230.204,-101.621,-36.194,179.535,5.283,149.057
C03158=1230.199,-101.370,-36.204,179.538,5.283,149.056
C03159=1230.193,-101.121,-36.215,179.540,5.283,149.055
C03160=1230.187,-100.850,-36.227,179.543,5.283,149.055
C03161=1230.182,-100.579,-36.238,179.546,5.283,149.054
C03162=1230.176,-100.308,-36.250,179.548,5.283,149.053
C03163=1230.170,-100.037,-36.261,179.551,5.283,149.052
C03164=1230.165,-99.788,-36.272,179.553,5.283,149.052
C03165=1230.160,-99.538,-36.283,179.556,5.283,149.051
C03166=1230.155,-99.287,-36.293,179.558,5.283,149.050
C03167=1230.149,-99.038,-36.304,179.560,5.283,149.049
C03168=1230.144,-98.788,-36.315,179.563,5.283,149.049
C03169=1230.139,-98.539,-36.325,179.565,5.283,149.048
C03170=1230.134,-98.289,-36.336,179.567,5.283,149.047
C03171=1230.129,-98.039,-36.347,179.570,5.284,149.047
C03172=1230.124,-97.789,-36.357,179.572,5.284,149.046
C03173=1230.118,-97.540,-36.368,179.574,5.284,149.045
C03174=1230.113,-97.290,-36.379,179.576,5.284,149.045
C03175=1230.108,-97.041,-36.390,179.578,5.283,149.044
C03176=1230.103,-96.791,-36.400,179.581,5.284,149.043
C03177=1230.097,-96.541,-36.410,179.583,5.283,149.043
C03178=1230.093,-96.292,-36.422,179.586,5.284,149.042
C03179=1230.087,-96.041,-36.433,179.588,5.283,149.041
C03180=1230.082,-95.792,-36.444,179.591,5.284,149.040
C03181=1230.077,-95.542,-36.454,179.593,5.284,149.040
C03182=1230.071,-95.292,-36.464,179.595,5.284,149.039
C03183=1230.066,-95.043,-36.476,179.597,5.284,149.038
C03184=1230.061,-94.793,-36.486,179.600,5.284,149.038
C03185=1230.056,-94.544,-36.497,179.602,5.284,149.037
C03186=1230.051,-94.293,-36.508,179.605,5.284,149.036
C03187=1230.046,-94.044,-36.519,179.607,5.284,149.035
C03188=1230.040,-93.794,-36.530,179.610,5.284,149.035
C03189=1230.035,-93.545,-36.541,179.612,5.284,149.034
C03190=1230.030,-93.295,-36.551,179.614,5.284,149.033
C03191=1230.025,-93.045,-36.563,179.617,5.284,149.033
C03192=1230.019,-92.796,-36.573,179.619,5.284,149.032
C03193=1230.015,-92.546,-36.584,179.621,5.285,149.031
C03194=1230.008,-92.296,-36.595,179.623,5.285,149.031
C03195=1230.004,-92.046,-36.606,179.626,5.285,149.030
C03196=1229.999,-91.796,-36.617,179.628,5.285,149.029
C03197=1229.993,-91.547,-36.628,179.630,5.285,149.029
C03198=1229.988,-91.297,-36.638,179.633,5.285,149.028
C03199=1229.983,-91.048,-36.649,179.635,5.285,149.027
C03200=1229.977,-90.798,-36.660,179.638,5.285,149.026
C03201=1229.973,-90.548,-36.672,179.640,5.285,149.026
C03202=1229.967,-90.298,-36.682,179.643,5.285,149.025
C03203=1229.962,-90.049,-36.693,179.645,5.285,149.024
C03204=1229.957,-89.799,-36.705,179.647,5.285,149.024
C03205=1229.951,-89.549,-36.715,179.649,5.285,149.023
C03206=1229.947,-89.300,-36.727,179.652,5.286,149.022
C03207=1229.942,-89.049,-36.737,179.654,5.285,149.021
C03208=1229.936,-88.801,-36.748,179.657,5.286,149.021
C03209=1229.931,-88.551,-36.760,179.659,5.285,149.020
C03210=1229.926,-88.300,-36.771,179.661,5.285,149.019
C03211=1229.921,-88.051,-36.782,179.664,5.285,149.019
C03212=1229.916,-87.801,-36.792,179.666,5.285,149.018
C03213=1229.910,-87.551,-36.804,179.668,5.285,149.017
C03214=1229.905,-87.302,-36.815,179.671,5.285,149.016
C03215=1229.900,-87.052,-36.826,179.673,5.286,149.016
C03216=1229.895,-86.802,-36.837,179.675,5.285,149.015
C03217=1229.889,-86.553,-36.848,179.678,5.286,149.014
C03218=1229.884,-86.303,-36.859,179.680,5.285,149.014
C03219=1229.880,-86.053,-36.870,179.683,5.286,149.013
C03220=1229.874,-85.804,-36.882,179.685,5.285,149.012
C03221=1229.869,-85.554,-36.892,179.688,5.286,149.011
C03222=1229.864,-85.304,-36.904,179.690,5.285,149.011
C03223=1229.858,-85.054,-36.915,179.692,5.286,149.010
C03224=1229.853,-84.805,-36.926,179.694,5.286,149.009
C03225=1229.848,-84.555,-36.937,179.697,5.286,149.009
C03226=1229.843,-84.305,-36.948,179.699,5.286,149.008
C03227=1229.837,-84.056,-36.960,179.701,5.287,149.007
C03228=1229.833,-83.807,-36.971,179.703,5.286,149.007
C03229=1229.828,-83.556,-36.982,179.706,5.287,149.006
C03230=1229.822,-83.306,-36.994,179.708,5.286,149.005
C03231=1229.817,-83.058,-37.004,179.711,5.287,149.005
C03232=1229.812,-82.808,-37.016,179.713,5.286,149.004
C03233=1229.807,-82.557,-37.027,179.716,5.287,149.003
C03234=1229.802,-82.308,-37.038,179.718,5.287,149.002
C03235=1229.796,-82.058,-37.050,179.720,5.287,149.002
C03236=1229.791,-81.809,-37.061,179.722,5.287,149.001
C03237=1229.786,-81.559,-37.072,179.725,5.287,149.000
C03238=1229.781,-81.309,-37.083,179.727,5.287,149.000
C03239=1229.775,-81.060,-37.094,179.730,5.287,148.999
C03240=1229.770,-80.810,-37.106,179.733,5.288,148.998
C03241=1229.765,-80.560,-37.118,179.735,5.287,148.997
C03242=1229.761,-80.311,-37.129,179.737,5.288,148.997
C03243=1229.755,-80.061,-37.140,179.739,5.287,148.996
C03244=1229.750,-79.811,-37.151,179.742,5.288,148.995
C03245=1229.744,-79.561,-37.163,179.744,5.288,148.995
C03246=1229.739,-79.311,-37.174,179.747,5.288,148.994
C03247=1229.735,-79.062,-37.185,179.749,5.288,148.993
C03248=1229.729,-78.813,-37.197,179.752,5.288,148.993
C03249=1229.724,-78.563,-37.208,179.754,5.288,148.992
C03250=1229.719,-78.313,-37.220,179.756,5.288,148.991
C03251=1229.714,-78.063,-37.231,179.758,5.288,148.990
C03252=1229.708,-77.813,-37.243,179.761,5.288,148.990
C03253=1229.703,-77.564,-37.253,179.763,5.288,148.989
C03254=1229.697,-77.314,-37.265,179.766,5.288,148.988
C03255=1229.693,-77.064,-37.277,179.768,5.288,148.988
C03256=1229.687,-76.814,-37.289,179.771,5.289,148.987
C03257=1229.683,-76.565,-37.300,179.773,5.288,148.986
C03258=1229.677,-76.316,-37.311,179.775,5.289,148.985
C03259=1229.672,-76.066,-37.323,179.778,5.288,148.985
C03260=1229.667,-75.816,-37.335,179.780,5.289,148.984
C03261=1229.662,-75.566,-37.346,179.782,5.288,148.983
C03262=1229.656,-75.316,-37.358,179.785,5.289,148.983
C03263=1229.652,-75.067,-37.369,179.787,5.289,148.982
C03264=1229.646,-74.797,-37.382,179.790,5.289,148.981
C03265=1229.640,-74.526,-37.394,179.793,5.289,148.980
C03266=1229.634,-74.257,-37.406,179.795,5.289,148.980
C03267=1229.629,-73.986,-37.419,179.798,5.289,148.979
C03268=1229.624,-73.736,-37.430,179.800,5.289,148.978
C03269=1229.619,-73.486,-37.442,179.802,5.289,148.977
C03270=1229.613,-73.236,-37.454,179.804,5.289,148.977
C03271=1229.608,-72.986,-37.465,179.807,5.289,148.976
C03272=1229.603,-72.738,-37.477,179.809,5.289,148.975
C03273=1229.598,-72.488,-37.489,179.812,5.290,148.975
C03274=1229.593,-72.238,-37.500,179.815,5.290,148.974
C03275=1229.588,-71.989,-37.512,179.817,5.290,148.973
C03276=1229.582,-71.739,-37.524,179.819,5.290,148.972
C03277=1229.577,-71.489,-37.536,179.821,5.290,148.972
C03278=1229.572,-71.239,-37.547,179.824,5.290,148.971
C03279=1229.567,-70.989,-37.559,179.826,5.290,148.970
C03280=1229.562,-70.740,-37.570,179.829,5.290,148.970
C03281=1229.556,-70.490,-37.581,179.831,5.290,148.969
C03282=1229.551,-70.240,-37.593,179.834,5.291,148.968
C03283=1229.546,-69.991,-37.605,179.836,5.290,148.967
C03284=1229.541,-69.742,-37.617,179.838,5.291,148.967
C03285=1229.536,-69.492,-37.629,179.840,5.290,148.966
C03286=1229.531,-69.242,-37.640,179.843,5.291,148.965
C03287=1229.525,-68.992,-37.652,179.845,5.290,148.965
C03288=1229.521,-68.742,-37.664,179.848,5.291,148.964
C03289=1229.515,-68.492,-37.676,179.850,5.291,148.963
C03290=1229.510,-68.243,-37.688,179.853,5.291,148.963
C03291=1229.505,-67.993,-37.699,179.855,5.291,148.962
C03292=1229.499,-67.744,-37.711,179.857,5.291,148.961
C03293=1229.494,-67.494,-37.723,179.860,5.292,148.960
C03294=1229.489,-67.245,-37.734,179.862,5.291,148.960
C03295=1229.484,-66.995,-37.747,179.865,5.292,148.959
C03296=1229.479,-66.745,-37.759,179.867,5.291,148.958
C03297=1229.474,-66.496,-37.770,179.870,5.292,148.958
C03298=1229.469,-66.246,-37.782,179.872,5.292,148.957
C03299=1229.464,-65.997,-37.794,179.874,5.292,148.956
C03300=1229.459,-65.747,-37.806,179.876,5.292,148.955
C03301=1229.453,-65.497,-37.818,179.879,5.292,148.955
C03302=1229.448,-65.247,-37.829,179.881,5.292,148.954
C03303=1229.443,-64.998,-37.842,179.884,5.292,148.953
C03304=1229.438,-64.748,-37.853,179.887,5.293,148.953
C03305=1229.433,-64.498,-37.865,179.889,5.292,148.952
C03306=1229.427,-64.248,-37.877,179.891,5.293,148.951
C03307=1229.423,-63.999,-37.889,179.893,5.293,148.951
C03308=1229.417,-63.749,-37.901,179.896,5.293,148.950
C03309=1229.412,-63.499,-37.913,179.898,5.293,148.949
C03310=1229.407,-63.250,-37.925,179.901,5.293,148.948
C03311=1229.402,-63.000,-37.937,179.903,5.293,148.948
C03312=1229.397,-62.750,-37.949,179.906,5.293,148.947
C03313=1229.392,-62.501,-37.961,179.908,5.293,148.946
C03314=1229.386,-62.251,-37.973,179.910,5.293,148.946
C03315=1229.381,-62.001,-37.985,179.912,5.293,148.945
C03316=1229.376,-61.752,-37.997,179.915,5.294,148.944
C03317=1229.371,-61.502,-38.009,179.918,5.294,148.943
C03318=1229.366,-61.253,-38.021,179.920,5.294,148.943
C03319=1229.360,-61.003,-38.033,179.923,5.294,148.942
C03320=1229.356,-60.753,-38.045,179.925,5.294,148.941
C03321=1229.351,-60.504,-38.057,179.927,5.294,148.941
C03322=1229.345,-60.254,-38.069,179.929,5.294,148.940
C03323=1229.340,-60.005,-38.082,179.932,5.294,148.939
C03324=1229.335,-59.755,-38.094,179.934,5.294,148.939
C03325=1229.329,-59.505,-38.106,179.937,5.294,148.938
C03326=1229.325,-59.256,-38.118,179.940,5.295,148.937
C03327=1229.319,-59.006,-38.129,179.942,5.294,148.936
C03328=1229.315,-58.756,-38.142,179.945,5.295,148.935
C03329=1229.309,-58.506,-38.154,179.947,5.294,148.935
C03330=1229.304,-58.257,-38.167,179.949,5.295,148.934
C03331=1229.299,-58.007,-38.179,179.952,5.295,148.933
C03332=1229.295,-57.758,-38.191,179.954,5.295,148.933
C03333=1229.289,-57.508,-38.203,179.956,5.295,148.932
C03334=1229.284,-57.259,-38.215,179.959,5.295,148.931
C03335=1229.279,-57.009,-38.227,179.962,5.296,148.931
C03336=1229.273,-56.759,-38.240,179.964,5.295,148.930
C03337=1229.268,-56.509,-38.252,179.966,5.296,148.929
C03338=1229.263,-56.260,-38.264,179.968,5.296,148.928
C03339=1229.257,-56.010,-38.276,179.971,5.296,148.928
C03340=1229.254,-55.760,-38.288,179.973,5.296,148.927
C03341=1229.248,-55.511,-38.300,179.976,5.296,148.926
C03342=1229.243,-55.261,-38.313,179.978,5.296,148.926
C03343=1229.238,-55.011,-38.325,179.981,5.296,148.925
C03344=1229.233,-54.762,-38.337,179.983,5.297,148.924
C03345=1229.227,-54.513,-38.350,179.985,5.296,148.924
C03346=1229.222,-54.263,-38.362,179.988,5.297,148.923
C03347=1229.217,-54.013,-38.375,179.990,5.297,148.922
C03348=1229.212,-53.763,-38.387,179.993,5.297,148.921
C03349=1229.207,-53.513,-38.399,179.995,5.297,148.921
C03350=1229.201,-53.263,-38.411,179.998,5.297,148.920
C03351=1229.196,-53.014,-38.424,-180.000,5.298,148.919
C03352=1229.191,-52.765,-38.436,-179.998,5.297,148.919
C03353=1229.186,-52.515,-38.448,-179.995,5.298,148.918
C03354=1229.181,-52.266,-38.461,-179.993,5.298,148.917
C03355=1229.176,-52.016,-38.474,-179.990,5.298,148.916
C03356=1229.171,-51.766,-38.486,-179.988,5.298,148.916
C03357=1229.166,-51.516,-38.498,-179.985,5.298,148.915
C03358=1229.160,-51.267,-38.511,-179.983,5.299,148.914
C03359=1229.155,-51.017,-38.523,-179.981,5.298,148.914
C03360=1229.150,-50.768,-38.535,-179.978,5.299,148.913
C03361=1229.145,-50.518,-38.548,-179.976,5.299,148.912
C03362=1229.140,-50.268,-38.560,-179.973,5.299,148.912
C03363=1229.135,-50.018,-38.573,-179.971,5.299,148.911
C03364=1229.130,-49.769,-38.586,-179.969,5.299,148.910
C03365=1229.124,-49.519,-38.597,-179.966,5.300,148.909
C03366=1229.120,-49.269,-38.610,-179.964,5.299,148.909
C03367=1229.115,-49.020,-38.623,-179.961,5.300,148.908
C03368=1229.109,-48.751,-38.636,-179.959,5.299,148.907
C03369=1229.104,-48.481,-38.649,-179.956,5.300,148.906
C03370=1229.098,-48.210,-38.664,-179.953,5.300,148.906
C03371=1229.092,-47.941,-38.677,-179.951,5.301,148.905
C03372=1229.088,-47.691,-38.690,-179.948,5.300,148.904
C03373=1229.082,-47.441,-38.702,-179.945,5.300,148.903
C03374=1229.077,-47.192,-38.714,-179.943,5.300,148.903
C03375=1229.072,-46.943,-38.727,-179.941,5.300,148.902
C03376=1229.067,-46.694,-38.740,-179.938,5.300,148.901
C03377=1229.061,-46.443,-38.752,-179.936,5.301,148.901
C03378=1229.056,-46.193,-38.765,-179.933,5.301,148.900
C03379=1229.051,-45.944,-38.778,-179.931,5.301,148.899
C03380=1229.046,-45.695,-38.790,-179.928,5.301,148.898
C03381=1229.042,-45.445,-38.803,-179.926,5.301,148.898
C03382=1229.036,-45.195,-38.816,-179.924,5.301,148.897
C03383=1229.031,-44.945,-38.828,-179.921,5.302,148.896
C03384=1229.026,-44.696,-38.840,-179.919,5.302,148.896
C03385=1229.021,-44.446,-38.854,-179.916,5.302,148.895
C03386=1229.016,-44.196,-38.866,-179.914,5.302,148.894
C03387=1229.010,-43.947,-38.879,-179.911,5.302,148.894
C03388=1229.005,-43.698,-38.892,-179.909,5.303,148.893
C03389=1229.001,-43.448,-38.905,-179.907,5.302,148.892
C03390=1228.996,-43.198,-38.917,-179.904,5.303,148.891
C03391=1228.990,-42.948,-38.929,-179.902,5.303,148.891
C03392=1228.984,-42.699,-38.942,-179.899,5.303,148.890
C03393=1228.980,-42.449,-38.955,-179.897,5.303,148.889
C03394=1228.975,-42.200,-38.968,-179.895,5.303,148.889
C03395=1228.970,-41.950,-38.980,-179.892,5.304,148.888
C03396=1228.965,-41.700,-38.993,-179.890,5.303,148.887
C03397=1228.959,-41.451,-39.007,-179.887,5.304,148.887
C03398=1228.954,-41.201,-39.019,-179.885,5.304,148.886
C03399=1228.950,-40.951,-39.032,-179.882,5.304,148.885
C03400=1228.944,-40.702,-39.045,-179.880,5.305,148.884
C03401=1228.939,-40.453,-39.057,-179.878,5.304,148.884
C03402=1228.933,-40.203,-39.071,-179.875,5.305,148.883
C03403=1228.929,-39.953,-39.083,-179.873,5.304,148.882
C03404=1228.924,-39.704,-39.096,-179.870,5.305,148.882
C03405=1228.919,-39.454,-39.109,-179.868,5.305,148.881
C03406=1228.913,-39.204,-39.122,-179.866,5.305,148.880
C03407=1228.908,-38.955,-39.135,-179.863,5.306,148.880
C03408=1228.903,-38.705,-39.147,-179.861,5.305,148.879
C03409=1228.899,-38.455,-39.160,-179.858,5.305,148.878
C03410=1228.893,-38.206,-39.174,-179.855,5.306,148.877
C03411=1228.888,-37.956,-39.186,-179.853,5.306,148.876
C03412=1228.883,-37.706,-39.199,-179.850,5.306,148.876
C03413=1228.878,-37.457,-39.212,-179.848,5.307,148.875
C03414=1228.873,-37.207,-39.225,-179.845,5.306,148.874
C03415=1228.868,-36.957,-39.238,-179.843,5.307,148.874
C03416=1228.862,-36.708,-39.251,-179.841,5.306,148.873
C03417=1228.858,-36.458,-39.265,-179.838,5.307,148.872
C03418=1228.852,-36.209,-39.277,-179.835,5.307,148.872
C03419=1228.847,-35.960,-39.290,-179.833,5.307,148.871
C03420=1228.842,-35.709,-39.304,-179.831,5.308,148.870
C03421=1228.837,-35.460,-39.316,-179.829,5.307,148.869
C03422=1228.832,-35.211,-39.329,-179.826,5.308,148.869
C03423=1228.827,-34.960,-39.342,-179.823,5.308,148.868
C03424=1228.821,-34.711,-39.355,-179.821,5.308,148.867
C03425=1228.817,-34.462,-39.369,-179.818,5.308,148.867
C03426=1228.811,-34.212,-39.382,-179.816,5.309,148.866
C03427=1228.806,-33.963,-39.394,-179.814,5.309,148.865
C03428=1228.802,-33.713,-39.407,-179.811,5.309,148.865
C03429=1228.796,-33.463,-39.421,-179.809,5.309,148.864
C03430=1228.791,-33.213,-39.434,-179.806,5.309,148.863
C03431=1228.786,-32.964,-39.447,-179.804,5.310,148.862
C03432=1228.781,-32.715,-39.460,-179.802,5.309,148.862
C03433=1228.776,-32.465,-39.473,-179.799,5.310,148.861
C03434=1228.770,-32.215,-39.486,-179.797,5.310,148.860
C03435=1228.766,-31.966,-39.500,-179.794,5.310,148.860
C03436=1228.760,-31.716,-39.513,-179.792,5.311,148.859
C03437=1228.756,-31.466,-39.526,-179.789,5.310,148.858
C03438=1228.751,-31.217,-39.539,-179.787,5.311,148.858
C03439=1228.746,-30.967,-39.553,-179.784,5.311,148.857
C03440=1228.740,-30.718,-39.566,-179.782,5.311,148.856
C03441=1228.735,-30.468,-39.579,-179.779,5.312,148.855
C03442=1228.730,-30.218,-39.592,-179.777,5.312,148.855
C03443=1228.724,-29.969,-39.606,-179.775,5.312,148.854
C03444=1228.720,-29.719,-39.619,-179.772,5.312,148.853
C03445=1228.715,-29.470,-39.631,-179.769,5.312,148.852
C03446=1228.710,-29.220,-39.645,-179.767,5.312,148.852
C03447=1228.705,-28.971,-39.658,-179.764,5.313,148.851
C03448=1228.699,-28.720,-39.672,-179.762,5.312,148.850
C03449=1228.695,-28.472,-39.685,-179.759,5.313,148.850
C03450=1228.689,-28.221,-39.699,-179.757,5.313,148.849
C03451=1228.684,-27.972,-39.711,-179.755,5.313,148.848
C03452=1228.679,-27.722,-39.725,-179.752,5.313,148.848
C03453=1228.674,-27.473,-39.738,-179.750,5.313,148.847
C03454=1228.669,-27.223,-39.752,-179.747,5.314,148.846
C03455=1228.664,-26.974,-39.765,-179.745,5.314,148.845
C03456=1228.659,-26.724,-39.778,-179.742,5.314,148.845
C03457=1228.654,-26.474,-39.791,-179.740,5.314,148.844
C03458=1228.649,-26.225,-39.805,-179.737,5.315,148.843
C03459=1228.644,-25.975,-39.818,-179.735,5.314,148.843
C03460=1228.639,-25.726,-39.832,-179.732,5.315,148.842
C03461=1228.634,-25.476,-39.845,-179.730,5.315,148.841
C03462=1228.629,-25.227,-39.859,-179.728,5.315,148.841
C03463=1228.624,-24.977,-39.872,-179.725,5.316,148.840
C03464=1228.618,-24.727,-39.885,-179.722,5.316,148.839
C03465=1228.613,-24.478,-39.899,-179.720,5.316,148.839
C03466=1228.608,-24.228,-39.912,-179.718,5.316,148.838
C03467=1228.603,-23.979,-39.926,-179.715,5.317,148.837
C03468=1228.598,-23.729,-39.939,-179.713,5.317,148.836
C03469=1228.593,-23.480,-39.953,-179.710,5.317,148.836
C03470=1228.588,-23.230,-39.966,-179.708,5.317,148.835
C03471=1228.583,-22.980,-39.980,-179.705,5.317,148.834
C03472=1228.577,-22.711,-39.995,-179.703,5.318,148.834
C03473=1228.572,-22.442,-40.008,-179.700,5.318,148.833
C03474=1228.567,-22.172,-40.023,-179.698,5.318,148.832
C03475=1228.561,-21.903,-40.038,-179.695,5.318,148.831
C03476=1228.555,-21.653,-40.052,-179.692,5.319,148.831
C03477=1228.551,-21.404,-40.065,-179.690,5.319,148.830
C03478=1228.546,-21.155,-40.079,-179.687,5.319,148.829
C03479=1228.540,-20.904,-40.093,-179.685,5.319,148.829
C03480=1228.535,-20.656,-40.106,-179.682,5.320,148.828
C03481=1228.530,-20.405,-40.120,-179.680,5.320,148.827
C03482=1228.525,-20.156,-40.134,-179.677,5.320,148.826
C03483=1228.520,-19.906,-40.147,-179.675,5.321,148.826
C03484=1228.515,-19.657,-40.161,-179.673,5.320,148.825
C03485=1228.510,-19.408,-40.175,-179.670,5.321,148.824
C03486=1228.505,-19.158,-40.188,-179.667,5.321,148.824
C03487=1228.500,-18.908,-40.202,-179.665,5.321,148.823
C03488=1228.494,-18.658,-40.215,-179.662,5.321,148.822
C03489=1228.490,-18.409,-40.229,-179.659,5.322,148.821
C03490=1228.485,-18.159,-40.243,-179.657,5.321,148.821
C03491=1228.479,-17.910,-40.256,-179.655,5.322,148.820
C03492=1228.475,-17.660,-40.270,-179.652,5.322,148.819
C03493=1228.469,-17.411,-40.284,-179.650,5.322,148.819
C03494=1228.464,-17.161,-40.297,-179.647,5.323,148.818
C03495=1228.459,-16.911,-40.312,-179.645,5.323,148.817
C03496=1228.454,-16.662,-40.325,-179.643,5.323,148.817
C03497=1228.449,-16.412,-40.339,-179.640,5.323,148.816
C03498=1228.444,-16.162,-40.353,-179.637,5.324,148.815
C03499=1228.439,-15.914,-40.366,-179.635,5.323,148.814
C03500=1228.434,-15.664,-40.381,-179.633,5.324,148.814
C03501=1228.429,-15.414,-40.394,-179.630,5.325,148.813
C03502=1228.424,-15.165,-40.408,-179.628,5.324,148.812
C03503=1228.419,-14.915,-40.422,-179.625,5.325,148.812
C03504=1228.414,-14.665,-40.435,-179.622,5.325,148.811
C03505=1228.409,-14.416,-40.449,-179.620,5.325,148.810
C03506=1228.404,-14.166,-40.463,-179.618,5.325,148.810
C03507=1228.399,-13.917,-40.478,-179.615,5.326,148.809
C03508=1228.394,-13.668,-40.491,-179.613,5.326,148.808
C03509=1228.389,-13.417,-40.505,-179.610,5.326,148.807
C03510=1228.384,-13.168,-40.519,-179.608,5.327,148.807
C03511=1228.378,-12.919,-40.533,-179.606,5.326,148.806
C03512=1228.373,-12.669,-40.547,-179.603,5.327,148.805
C03513=1228.369,-12.420,-40.561,-179.600,5.327,148.805
C03514=1228.363,-12.170,-40.574,-179.598,5.327,148.804
C03515=1228.358,-11.920,-40.588,-179.596,5.328,148.803
C03516=1228.353,-11.671,-40.602,-179.593,5.328,148.803
C03517=1228.348,-11.421,-40.617,-179.591,5.328,148.802
C03518=1228.343,-11.172,-40.631,-179.588,5.328,148.801
C03519=1228.338,-10.923,-40.644,-179.586,5.329,148.801
C03520=1228.333,-10.672,-40.658,-179.583,5.329,148.800
C03521=1228.328,-10.422,-40.672,-179.581,5.329,148.799
C03522=1228.323,-10.173,-40.686,-179.578,5.330,148.798
C03523=1228.318,-9.924,-40.700,-179.575,5.330,148.798
C03524=1228.313,-9.674,-40.715,-179.573,5.330,148.797
C03525=1228.308,-9.424,-40.729,-179.571,5.330,148.796
C03526=1228.303,-9.176,-40.742,-179.568,5.331,148.796
C03527=1228.298,-8.926,-40.757,-179.566,5.331,148.795
C03528=1228.293,-8.676,-40.771,-179.563,5.331,148.794
C03529=1228.288,-8.426,-40.785,-179.561,5.332,148.794
C03530=1228.283,-8.177,-40.799,-179.558,5.332,148.793
C03531=1228.278,-7.928,-40.813,-179.556,5.332,148.792
C03532=1228.272,-7.677,-40.827,-179.553,5.332,148.792
C03533=1228.267,-7.428,-40.841,-179.551,5.333,148.791
C03534=1228.262,-7.179,-40.855,-179.549,5.333,148.790
C03535=1228.257,-6.929,-40.869,-179.546,5.333,148.789
C03536=1228.252,-6.679,-40.884,-179.543,5.334,148.789
C03537=1228.247,-6.430,-40.898,-179.541,5.333,148.788
C03538=1228.243,-6.180,-40.912,-179.539,5.334,148.787
C03539=1228.237,-5.931,-40.925,-179.536,5.334,148.787
C03540=1228.232,-5.681,-40.940,-179.533,5.335,148.786
C03541=1228.227,-5.432,-40.954,-179.531,5.335,148.785
C03542=1228.223,-5.183,-40.969,-179.528,5.335,148.785
C03543=1228.218,-4.933,-40.983,-179.526,5.336,148.784
C03544=1228.212,-4.684,-40.997,-179.524,5.335,148.783
C03545=1228.207,-4.434,-41.011,-179.521,5.336,148.783
C03546=1228.202,-4.185,-41.026,-179.518,5.336,148.782
C03547=1228.197,-3.935,-41.040,-179.516,5.337,148.781
C03548=1228.192,-3.685,-41.054,-179.514,5.337,148.781
C03549=1228.187,-3.435,-41.069,-179.511,5.337,148.780
C03550=1228.182,-3.186,-41.082,-179.508,5.338,148.779
C03551=1228.177,-2.937,-41.097,-179.506,5.337,148.778
C03552=1228.172,-2.687,-41.111,-179.504,5.338,148.778
C03553=1228.167,-2.437,-41.125,-179.501,5.338,148.777
C03554=1228.162,-2.188,-41.140,-179.498,5.339,148.776
C03555=1228.157,-1.938,-41.155,-179.496,5.339,148.776
C03556=1228.151,-1.689,-41.169,-179.494,5.339,148.775
C03557=1228.146,-1.439,-41.183,-179.491,5.340,148.774
C03558=1228.141,-1.190,-41.198,-179.489,5.339,148.774
C03559=1228.136,-0.940,-41.212,-179.486,5.340,148.773
C03560=1228.132,-0.691,-41.227,-179.484,5.340,148.772
C03561=1228.127,-0.441,-41.241,-179.481,5.341,148.772
C03562=1228.122,-0.191,-41.255,-179.479,5.341,148.771
C03563=1228.117,0.058,-41.270,-179.476,5.341,148.770
C03564=1228.111,0.307,-41.284,-179.474,5.342,148.769
C03565=1228.106,0.556,-41.299,-179.471,5.342,148.769
C03566=1228.101,0.806,-41.313,-179.469,5.342,148.768
C03567=1228.096,1.056,-41.328,-179.466,5.342,148.767
C03568=1228.091,1.306,-41.342,-179.464,5.343,148.767
C03569=1228.086,1.555,-41.356,-179.461,5.344,148.766
C03570=1228.081,1.805,-41.371,-179.459,5.343,148.765
C03571=1228.076,2.054,-41.386,-179.456,5.344,148.765
C03572=1228.071,2.304,-41.400,-179.453,5.344,148.764
C03573=1228.066,2.554,-41.414,-179.451,5.344,148.763
C03574=1228.062,2.803,-41.429,-179.449,5.345,148.763
C03575=1228.055,3.052,-41.444,-179.446,5.345,148.762
C03576=1228.050,3.321,-41.459,-179.443,5.345,148.761
C03577=1228.045,3.590,-41.475,-179.440,5.346,148.760
C03578=1228.040,3.858,-41.491,-179.438,5.346,148.760
C03579=1228.034,4.128,-41.506,-179.436,5.346,148.759
C03580=1228.029,4.377,-41.521,-179.433,5.347,148.758
C03581=1228.024,4.627,-41.536,-179.430,5.347,148.758
C03582=1228.019,4.877,-41.550,-179.428,5.348,148.757
C03583=1228.015,5.126,-41.565,-179.426,5.347,148.756
C03584=1228.009,5.376,-41.580,-179.423,5.348,148.755
C03585=1228.004,5.625,-41.595,-179.420,5.348,148.755
C03586=1227.999,5.875,-41.609,-179.418,5.349,148.754
C03587=1227.994,6.124,-41.623,-179.416,5.349,148.753
C03588=1227.990,6.373,-41.638,-179.413,5.349,148.753
C03589=1227.984,6.623,-41.653,-179.410,5.350,148.752
C03590=1227.979,6.873,-41.668,-179.408,5.350,148.751
C03591=1227.974,7.122,-41.682,-179.405,5.350,148.751
C03592=1227.970,7.372,-41.697,-179.403,5.350,148.750
C03593=1227.964,7.621,-41.712,-179.400,5.351,148.749
C03594=1227.959,7.871,-41.727,-179.398,5.351,148.749
C03595=1227.955,8.120,-41.742,-179.395,5.351,148.748
C03596=1227.950,8.370,-41.756,-179.393,5.352,148.747
C03597=1227.944,8.619,-41.771,-179.390,5.352,148.747
C03598=1227.939,8.869,-41.786,-179.388,5.353,148.746
C03599=1227.935,9.118,-41.801,-179.385,5.353,148.745
C03600=1227.929,9.368,-41.816,-179.383,5.353,148.744
C03601=1227.924,9.617,-41.831,-179.380,5.354,148.744
C03602=1227.919,9.867,-41.845,-179.377,5.354,148.743
C03603=1227.915,10.116,-41.860,-179.375,5.355,148.742
C03604=1227.909,10.366,-41.875,-179.373,5.354,148.742
C03605=1227.904,10.615,-41.890,-179.370,5.355,148.741
C03606=1227.899,10.865,-41.904,-179.367,5.355,148.740
C03607=1227.894,11.114,-41.920,-179.365,5.356,148.740
C03608=1227.889,11.364,-41.934,-179.363,5.356,148.739
C03609=1227.884,11.613,-41.949,-179.360,5.356,148.738
C03610=1227.879,11.863,-41.964,-179.357,5.357,148.738
C03611=1227.874,12.112,-41.979,-179.355,5.357,148.737
C03612=1227.869,12.362,-41.994,-179.352,5.358,148.736
C03613=1227.864,12.611,-42.009,-179.350,5.358,148.736
C03614=1227.859,12.860,-42.024,-179.347,5.358,148.735
C03615=1227.853,13.110,-42.038,-179.345,5.359,148.734
C03616=1227.849,13.359,-42.053,-179.342,5.359,148.734
C03617=1227.845,13.609,-42.069,-179.340,5.359,148.733
C03618=1227.839,13.859,-42.084,-179.337,5.359,148.732
C03619=1227.834,14.108,-42.099,-179.335,5.360,148.731
C03620=1227.829,14.358,-42.114,-179.332,5.360,148.731
C03621=1227.824,14.607,-42.129,-179.329,5.361,148.730
C03622=1227.819,14.857,-42.144,-179.327,5.361,148.729
C03623=1227.814,15.107,-42.158,-179.325,5.362,148.729
C03624=1227.809,15.356,-42.173,-179.323,5.362,148.728
C03625=1227.804,15.605,-42.189,-179.320,5.363,148.728
C03626=1227.799,15.854,-42.204,-179.318,5.362,148.727
C03627=1227.793,16.104,-42.219,-179.315,5.363,148.726
C03628=1227.789,16.354,-42.234,-179.313,5.364,148.726
C03629=1227.784,16.603,-42.250,-179.310,5.364,148.725
C03630=1227.779,16.853,-42.264,-179.307,5.365,148.724
C03631=1227.774,17.102,-42.279,-179.305,5.364,148.723
C03632=1227.769,17.352,-42.295,-179.303,5.365,148.723
C03633=1227.764,17.601,-42.310,-179.300,5.365,148.722
C03634=1227.758,17.851,-42.325,-179.297,5.366,148.721
C03635=1227.754,18.101,-42.340,-179.295,5.366,148.721
C03636=1227.749,18.350,-42.355,-179.293,5.366,148.720
C03637=1227.744,18.599,-42.370,-179.290,5.367,148.719
C03638=1227.739,18.849,-42.385,-179.287,5.367,148.719
C03639=1227.734,19.098,-42.400,-179.285,5.368,148.718
C03640=1227.729,19.348,-42.416,-179.282,5.368,148.717
C03641=1227.724,19.597,-42.431,-179.280,5.368,148.717
C03642=1227.719,19.847,-42.447,-179.277,5.369,148.716
C03643=1227.715,20.096,-42.462,-179.275,5.369,148.715
C03644=1227.709,20.346,-42.477,-179.272,5.370,148.715
C03645=1227.703,20.595,-42.492,-179.269,5.370,148.714
